C09146=1167.834,261.532,-67.033,-177.260,7.589,148.648
C09147=1167.838,261.283,-67.006,-177.262,7.587,148.648
C09148=1167.844,261.034,-66.978,-177.265,7.584,148.648
C09149=1167.847,260.786,-66.950,-177.268,7.581,148.649
C09150=1167.852,260.537,-66.922,-177.270,7.578,148.649
C09151=1167.856,260.290,-66.895,-177.273,7.575,148.649
C09152=1167.860,260.041,-66.867,-177.275,7.573,148.649
C09153=1167.865,259.792,-66.839,-177.278,7.570,148.649
C09154=1167.870,259.544,-66.811,-177.281,7.567,148.649
C09155=1167.874,259.296,-66.783,-177.284,7.564,148.649
C09156=1167.878,259.047,-66.756,-177.287,7.561,148.649
C09157=1167.883,258.799,-66.728,-177.289,7.559,148.649
C09158=1167.887,258.550,-66.701,-177.292,7.556,148.649
C09159=1167.891,258.302,-66.673,-177.295,7.553,148.649
C09160=1167.896,258.053,-66.645,-177.297,7.550,148.649
C09161=1167.900,257.805,-66.617,-177.299,7.548,148.650
C09162=1167.905,257.556,-66.590,-177.302,7.545,148.650
C09163=1167.909,257.309,-66.562,-177.305,7.542,148.650
C09164=1167.913,257.059,-66.535,-177.308,7.539,148.650
C09165=1167.917,256.811,-66.507,-177.310,7.537,148.650
C09166=1167.922,256.563,-66.480,-177.313,7.534,148.650
C09167=1167.926,256.314,-66.452,-177.316,7.531,148.650
C09168=1167.931,256.066,-66.425,-177.319,7.528,148.650
C09169=1167.935,255.818,-66.397,-177.321,7.526,148.650
C09170=1167.940,255.570,-66.370,-177.324,7.523,148.650
C09171=1167.944,255.320,-66.343,-177.326,7.520,148.650
C09172=1167.948,255.072,-66.315,-177.329,7.517,148.650
C09173=1167.953,254.824,-66.288,-177.331,7.515,148.651
C09174=1167.957,254.575,-66.260,-177.334,7.512,148.651
C09175=1167.961,254.327,-66.233,-177.337,7.510,148.651
C09176=1167.966,254.078,-66.205,-177.340,7.507,148.651
C09177=1167.970,253.830,-66.178,-177.342,7.505,148.651
C09178=1167.974,253.581,-66.150,-177.345,7.502,148.651
C09179=1167.979,253.333,-66.123,-177.348,7.499,148.651
C09180=1167.983,253.084,-66.096,-177.350,7.496,148.651
C09181=1167.988,252.836,-66.068,-177.353,7.494,148.651
C09182=1167.992,252.588,-66.041,-177.355,7.491,148.651
C09183=1167.996,252.339,-66.014,-177.359,7.488,148.652
C09184=1168.001,252.090,-65.987,-177.361,7.485,148.652
C09185=1168.005,251.842,-65.959,-177.364,7.483,148.652
C09186=1168.010,251.594,-65.932,-177.366,7.480,148.652
C09187=1168.014,251.346,-65.906,-177.369,7.477,148.652
C09188=1168.018,251.096,-65.878,-177.371,7.475,148.652
C09189=1168.023,250.848,-65.851,-177.375,7.472,148.652
C09190=1168.027,250.599,-65.824,-177.377,7.469,148.652
C09191=1168.032,250.352,-65.796,-177.380,7.466,148.652
C09192=1168.036,250.103,-65.769,-177.382,7.464,148.653
C09193=1168.041,249.855,-65.742,-177.385,7.461,148.653
C09194=1168.044,249.606,-65.715,-177.388,7.458,148.653
C09195=1168.049,249.357,-65.688,-177.390,7.457,148.653
C09196=1168.054,249.109,-65.661,-177.393,7.454,148.653
C09197=1168.058,248.860,-65.634,-177.396,7.451,148.653
C09198=1168.063,248.612,-65.607,-177.399,7.448,148.653
C09199=1168.067,248.364,-65.581,-177.401,7.446,148.653
C09200=1168.072,248.115,-65.553,-177.404,7.443,148.654
C09201=1168.076,247.866,-65.526,-177.407,7.440,148.654
C09202=1168.080,247.617,-65.499,-177.409,7.438,148.654
C09203=1168.084,247.369,-65.472,-177.412,7.435,148.654
C09204=1168.089,247.121,-65.445,-177.415,7.432,148.654
C09205=1168.094,246.872,-65.418,-177.417,7.430,148.654
C09206=1168.098,246.624,-65.391,-177.420,7.427,148.654
C09207=1168.102,246.376,-65.365,-177.423,7.424,148.654
C09208=1168.107,246.127,-65.338,-177.425,7.421,148.654
C09209=1168.111,245.879,-65.311,-177.428,7.419,148.655
C09210=1168.116,245.630,-65.284,-177.431,7.416,148.655
C09211=1168.120,245.382,-65.257,-177.434,7.413,148.655
C09212=1168.125,245.133,-65.231,-177.436,7.411,148.655
C09213=1168.129,244.884,-65.203,-177.439,7.408,148.655
C09214=1168.133,244.635,-65.177,-177.442,7.406,148.655
C09215=1168.138,244.387,-65.150,-177.444,7.404,148.655
C09216=1168.142,244.138,-65.123,-177.447,7.401,148.655
C09217=1168.146,243.890,-65.096,-177.449,7.398,148.656
C09218=1168.151,243.641,-65.070,-177.452,7.396,148.656
C09219=1168.155,243.393,-65.044,-177.455,7.393,148.656
C09220=1168.160,243.144,-65.016,-177.458,7.390,148.656
C09221=1168.164,242.896,-64.989,-177.460,7.388,148.656
C09222=1168.169,242.647,-64.964,-177.463,7.385,148.656
C09223=1168.173,242.399,-64.937,-177.466,7.382,148.656
C09224=1168.177,242.150,-64.910,-177.468,7.380,148.657
C09225=1168.182,241.901,-64.884,-177.471,7.377,148.657
C09226=1168.186,241.653,-64.857,-177.474,7.375,148.657
C09227=1168.191,241.405,-64.830,-177.476,7.372,148.657
C09228=1168.195,241.156,-64.803,-177.479,7.370,148.657
C09229=1168.200,240.907,-64.777,-177.482,7.367,148.657
C09230=1168.204,240.659,-64.750,-177.484,7.365,148.658
C09231=1168.208,240.410,-64.725,-177.487,7.362,148.658
C09232=1168.213,240.162,-64.698,-177.490,7.359,148.658
C09233=1168.217,239.913,-64.671,-177.493,7.357,148.658
C09234=1168.222,239.664,-64.645,-177.495,7.354,148.658
C09235=1168.227,239.417,-64.619,-177.497,7.352,148.658
C09236=1168.232,239.168,-64.592,-177.500,7.349,148.658
C09237=1168.235,238.919,-64.566,-177.503,7.346,148.659
C09238=1168.240,238.670,-64.540,-177.506,7.344,148.659
C09239=1168.244,238.422,-64.513,-177.508,7.341,148.659
C09240=1168.249,238.173,-64.487,-177.512,7.339,148.659
C09241=1168.253,237.925,-64.460,-177.514,7.337,148.659
C09242=1168.257,237.676,-64.434,-177.517,7.334,148.659
C09243=1168.262,237.428,-64.407,-177.520,7.331,148.659
C09244=1168.266,237.179,-64.382,-177.522,7.329,148.660
C09245=1168.271,236.930,-64.355,-177.525,7.326,148.660
C09246=1168.275,236.681,-64.329,-177.527,7.324,148.660
C09247=1168.280,236.411,-64.300,-177.530,7.321,148.660
C09248=1168.286,236.139,-64.272,-177.533,7.318,148.660
C09249=1168.290,235.867,-64.243,-177.536,7.316,148.660
C09250=1168.295,235.595,-64.214,-177.539,7.313,148.660
C09251=1168.299,235.347,-64.188,-177.542,7.310,148.661
C09252=1168.304,235.098,-64.162,-177.544,7.308,148.661
C09253=1168.309,234.849,-64.136,-177.547,7.305,148.661
C09254=1168.312,234.601,-64.109,-177.550,7.302,148.661
C09255=1168.317,234.352,-64.084,-177.553,7.300,148.661
C09256=1168.322,234.104,-64.058,-177.555,7.297,148.661
C09257=1168.326,233.855,-64.031,-177.558,7.295,148.662
C09258=1168.330,233.607,-64.005,-177.561,7.293,148.662
C09259=1168.335,233.358,-63.980,-177.563,7.290,148.662
C09260=1168.339,233.109,-63.953,-177.566,7.288,148.662
C09261=1168.344,232.861,-63.927,-177.569,7.285,148.662
C09262=1168.348,232.612,-63.902,-177.571,7.283,148.662
C09263=1168.353,232.363,-63.875,-177.574,7.280,148.663
C09264=1168.357,232.115,-63.849,-177.577,7.277,148.663
C09265=1168.361,231.866,-63.823,-177.580,7.275,148.663
C09266=1168.366,231.618,-63.798,-177.582,7.272,148.663
C09267=1168.370,231.369,-63.772,-177.585,7.270,148.663
C09268=1168.375,231.120,-63.745,-177.588,7.268,148.664
C09269=1168.380,230.871,-63.720,-177.591,7.265,148.664
C09270=1168.384,230.623,-63.694,-177.593,7.263,148.664
C09271=1168.389,230.375,-63.669,-177.596,7.260,148.664
C09272=1168.393,230.126,-63.642,-177.598,7.258,148.664
C09273=1168.398,229.877,-63.616,-177.602,7.255,148.664
C09274=1168.402,229.628,-63.590,-177.604,7.253,148.665
C09275=1168.407,229.380,-63.565,-177.606,7.250,148.665
C09276=1168.411,229.132,-63.539,-177.610,7.247,148.665
C09277=1168.415,228.883,-63.513,-177.612,7.245,148.665
C09278=1168.420,228.635,-63.488,-177.615,7.243,148.665
C09279=1168.424,228.386,-63.462,-177.617,7.241,148.665
C09280=1168.429,228.137,-63.436,-177.620,7.238,148.666
C09281=1168.433,227.888,-63.410,-177.623,7.236,148.666
C09282=1168.438,227.640,-63.385,-177.625,7.233,148.666
C09283=1168.442,227.391,-63.359,-177.628,7.231,148.666
C09284=1168.447,227.142,-63.333,-177.631,7.228,148.666
C09285=1168.451,226.894,-63.308,-177.634,7.225,148.666
C09286=1168.456,226.645,-63.282,-177.636,7.223,148.667
C09287=1168.460,226.397,-63.256,-177.639,7.220,148.667
C09288=1168.465,226.148,-63.231,-177.642,7.219,148.667
C09289=1168.469,225.899,-63.206,-177.645,7.216,148.667
C09290=1168.473,225.650,-63.180,-177.647,7.214,148.668
C09291=1168.478,225.402,-63.155,-177.650,7.211,148.668
C09292=1168.482,225.153,-63.129,-177.652,7.209,148.668
C09293=1168.487,224.904,-63.103,-177.655,7.206,148.668
C09294=1168.492,224.656,-63.078,-177.658,7.204,148.668
C09295=1168.496,224.408,-63.052,-177.661,7.202,148.669
C09296=1168.500,224.158,-63.027,-177.663,7.199,148.669
C09297=1168.505,223.910,-63.002,-177.666,7.197,148.669
C09298=1168.509,223.661,-62.976,-177.668,7.195,148.669
C09299=1168.514,223.413,-62.950,-177.672,7.192,148.669
C09300=1168.519,223.164,-62.925,-177.674,7.190,148.669
C09301=1168.523,222.915,-62.900,-177.677,7.187,148.670
C09302=1168.528,222.667,-62.874,-177.680,7.184,148.670
C09303=1168.532,222.418,-62.848,-177.682,7.182,148.670
C09304=1168.537,222.169,-62.824,-177.685,7.180,148.670
C09305=1168.541,221.920,-62.798,-177.687,7.178,148.670
C09306=1168.546,221.672,-62.772,-177.691,7.175,148.671
C09307=1168.550,221.423,-62.748,-177.693,7.173,148.671
C09308=1168.554,221.174,-62.722,-177.696,7.170,148.671
C09309=1168.559,220.926,-62.697,-177.698,7.168,148.671
C09310=1168.564,220.677,-62.672,-177.702,7.165,148.672
C09311=1168.568,220.429,-62.647,-177.704,7.163,148.672
C09312=1168.573,220.180,-62.621,-177.707,7.161,148.672
C09313=1168.577,219.931,-62.596,-177.709,7.159,148.672
C09314=1168.581,219.683,-62.571,-177.712,7.156,148.672
C09315=1168.586,219.433,-62.546,-177.715,7.154,148.673
C09316=1168.591,219.185,-62.521,-177.718,7.151,148.673
C09317=1168.595,218.936,-62.496,-177.720,7.149,148.673
C09318=1168.600,218.688,-62.470,-177.723,7.146,148.673
C09319=1168.604,218.439,-62.446,-177.725,7.144,148.673
C09320=1168.609,218.191,-62.420,-177.728,7.143,148.674
C09321=1168.613,217.941,-62.395,-177.731,7.140,148.674
C09322=1168.618,217.693,-62.370,-177.734,7.138,148.674
C09323=1168.622,217.444,-62.345,-177.736,7.135,148.674
C09324=1168.627,217.196,-62.320,-177.739,7.133,148.675
C09325=1168.631,216.946,-62.295,-177.742,7.130,148.675
C09326=1168.636,216.698,-62.270,-177.744,7.128,148.675
C09327=1168.640,216.449,-62.245,-177.747,7.125,148.675
C09328=1168.644,216.201,-62.220,-177.750,7.124,148.675
C09329=1168.649,215.952,-62.195,-177.753,7.121,148.675
C09330=1168.654,215.703,-62.170,-177.755,7.119,148.676
C09331=1168.658,215.454,-62.145,-177.758,7.116,148.676
C09332=1168.663,215.206,-62.120,-177.761,7.114,148.676
C09333=1168.668,214.958,-62.095,-177.764,7.111,148.676
C09334=1168.671,214.708,-62.071,-177.766,7.109,148.677
C09335=1168.677,214.460,-62.046,-177.768,7.107,148.677
C09336=1168.681,214.211,-62.020,-177.772,7.105,148.677
C09337=1168.685,213.963,-61.996,-177.774,7.103,148.677
C09338=1168.690,213.713,-61.971,-177.777,7.100,148.678
C09339=1168.695,213.464,-61.946,-177.780,7.098,148.678
C09340=1168.699,213.217,-61.922,-177.782,7.095,148.678
C09341=1168.703,212.967,-61.897,-177.785,7.094,148.678
C09342=1168.708,212.719,-61.872,-177.788,7.091,148.678
C09343=1168.712,212.469,-61.847,-177.791,7.089,148.679
C09344=1168.717,212.221,-61.822,-177.793,7.087,148.679
C09345=1168.722,211.973,-61.798,-177.796,7.084,148.679
C09346=1168.726,211.723,-61.773,-177.798,7.082,148.679
C09347=1168.730,211.475,-61.749,-177.801,7.079,148.680
C09348=1168.736,211.226,-61.724,-177.804,7.078,148.680
C09349=1168.739,210.977,-61.700,-177.807,7.075,148.680
C09350=1168.744,210.729,-61.674,-177.810,7.073,148.680
C09351=1168.749,210.458,-61.647,-177.812,7.070,148.680
C09352=1168.754,210.187,-61.621,-177.815,7.068,148.681
C09353=1168.759,209.917,-61.595,-177.818,7.065,148.681
C09354=1168.764,209.646,-61.568,-177.821,7.063,148.681
C09355=1168.768,209.398,-61.543,-177.824,7.061,148.682
C09356=1168.773,209.149,-61.519,-177.827,7.058,148.682
C09357=1168.777,208.900,-61.494,-177.829,7.056,148.682
C09358=1168.782,208.651,-61.470,-177.832,7.053,148.682
C09359=1168.787,208.403,-61.446,-177.835,7.051,148.682
C09360=1168.791,208.153,-61.421,-177.837,7.050,148.683
C09361=1168.796,207.905,-61.396,-177.840,7.047,148.683
C09362=1168.801,207.656,-61.372,-177.843,7.045,148.683
C09363=1168.805,207.408,-61.348,-177.846,7.042,148.684
C09364=1168.810,207.159,-61.323,-177.848,7.040,148.684
C09365=1168.814,206.910,-61.299,-177.851,7.038,148.684
C09366=1168.819,206.662,-61.275,-177.854,7.036,148.684
C09367=1168.824,206.413,-61.250,-177.856,7.034,148.684
C09368=1168.827,206.164,-61.225,-177.859,7.031,148.685
C09369=1168.833,205.915,-61.201,-177.862,7.029,148.685
C09370=1168.837,205.667,-61.177,-177.864,7.027,148.685
C09371=1168.841,205.418,-61.153,-177.868,7.024,148.686
C09372=1168.846,205.169,-61.128,-177.870,7.022,148.686
C09373=1168.850,204.920,-61.104,-177.872,7.021,148.686
C09374=1168.855,204.671,-61.080,-177.875,7.018,148.686
C09375=1168.860,204.423,-61.055,-177.878,7.016,148.686
C09376=1168.864,204.174,-61.031,-177.881,7.013,148.687
C09377=1168.868,203.925,-61.007,-177.883,7.011,148.687
C09378=1168.873,203.676,-60.982,-177.886,7.009,148.687
C09379=1168.878,203.427,-60.959,-177.889,7.007,148.688
C09380=1168.882,203.178,-60.934,-177.891,7.005,148.688
C09381=1168.887,202.930,-60.910,-177.894,7.003,148.688
C09382=1168.892,202.681,-60.886,-177.897,7.000,148.688
C09383=1168.896,202.433,-60.862,-177.900,6.998,148.688
C09384=1168.901,202.184,-60.838,-177.903,6.996,148.689
C09385=1168.905,201.934,-60.813,-177.905,6.993,148.689
C09386=1168.910,201.686,-60.789,-177.908,6.992,148.689
C09387=1168.914,201.437,-60.766,-177.911,6.989,148.690
C09388=1168.919,201.188,-60.742,-177.913,6.987,148.690
C09389=1168.924,200.940,-60.717,-177.916,6.985,148.690
C09390=1168.928,200.691,-60.694,-177.919,6.983,148.690
C09391=1168.932,200.442,-60.669,-177.921,6.980,148.691
C09392=1168.937,200.193,-60.645,-177.924,6.979,148.691
C09393=1168.941,199.944,-60.622,-177.927,6.976,148.691
C09394=1168.946,199.695,-60.597,-177.929,6.974,148.691
C09395=1168.951,199.446,-60.574,-177.932,6.972,148.692
C09396=1168.956,199.198,-60.550,-177.935,6.969,148.692
C09397=1168.960,198.950,-60.526,-177.937,6.967,148.692
C09398=1168.965,198.701,-60.502,-177.940,6.966,148.692
C09399=1168.968,198.451,-60.478,-177.943,6.963,148.693
C09400=1168.974,198.202,-60.454,-177.946,6.961,148.693
C09401=1168.978,197.954,-60.430,-177.948,6.959,148.693
C09402=1168.983,197.705,-60.407,-177.951,6.956,148.693
C09403=1168.987,197.456,-60.382,-177.954,6.954,148.694
C09404=1168.992,197.207,-60.359,-177.956,6.953,148.694
C09405=1168.996,196.959,-60.335,-177.959,6.950,148.694
C09406=1169.001,196.710,-60.312,-177.962,6.948,148.695
C09407=1169.006,196.461,-60.288,-177.965,6.946,148.695
C09408=1169.010,196.212,-60.264,-177.968,6.944,148.695
C09409=1169.015,195.964,-60.240,-177.970,6.942,148.695
C09410=1169.019,195.715,-60.217,-177.973,6.940,148.696
C09411=1169.024,195.465,-60.192,-177.976,6.937,148.696
C09412=1169.029,195.216,-60.168,-177.978,6.935,148.696
C09413=1169.033,194.967,-60.145,-177.981,6.933,148.697
C09414=1169.038,194.719,-60.121,-177.984,6.931,148.697
C09415=1169.042,194.470,-60.098,-177.986,6.929,148.697
C09416=1169.047,194.221,-60.074,-177.989,6.927,148.697
C09417=1169.051,193.972,-60.050,-177.992,6.924,148.698
C09418=1169.056,193.723,-60.027,-177.995,6.922,148.698
C09419=1169.061,193.474,-60.003,-177.997,6.920,148.698
C09420=1169.065,193.226,-59.979,-178.000,6.919,148.698
C09421=1169.070,192.977,-59.956,-178.003,6.916,148.699
C09422=1169.075,192.728,-59.933,-178.005,6.914,148.699
C09423=1169.079,192.479,-59.909,-178.008,6.912,148.699
C09424=1169.084,192.230,-59.885,-178.011,6.909,148.700
C09425=1169.088,191.982,-59.862,-178.013,6.907,148.700
C09426=1169.092,191.733,-59.839,-178.016,6.906,148.700
C09427=1169.097,191.484,-59.816,-178.019,6.903,148.700
C09428=1169.102,191.235,-59.792,-178.022,6.901,148.701
C09429=1169.106,190.986,-59.768,-178.024,6.899,148.701
C09430=1169.111,190.737,-59.745,-178.027,6.897,148.701
C09431=1169.116,190.489,-59.722,-178.030,6.895,148.702
C09432=1169.121,190.240,-59.699,-178.033,6.893,148.702
C09433=1169.126,189.991,-59.675,-178.035,6.891,148.702
C09434=1169.130,189.742,-59.651,-178.038,6.889,148.702
C09435=1169.135,189.493,-59.628,-178.041,6.886,148.703
C09436=1169.139,189.245,-59.605,-178.043,6.885,148.703
C09437=1169.143,188.996,-59.582,-178.046,6.883,148.703
C09438=1169.148,188.747,-59.558,-178.049,6.880,148.704
C09439=1169.153,188.498,-59.535,-178.052,6.878,148.704
C09440=1169.157,188.249,-59.512,-178.054,6.876,148.704
C09441=1169.162,187.999,-59.488,-178.056,6.874,148.704
C09442=1169.166,187.751,-59.465,-178.060,6.872,148.705
C09443=1169.171,187.502,-59.442,-178.062,6.870,148.705
C09444=1169.176,187.253,-59.419,-178.065,6.868,148.705
C09445=1169.181,187.004,-59.396,-178.067,6.866,148.706
C09446=1169.186,186.755,-59.372,-178.071,6.864,148.706
C09447=1169.189,186.507,-59.350,-178.073,6.862,148.706
C09448=1169.194,186.258,-59.326,-178.076,6.860,148.707
C09449=1169.199,186.009,-59.303,-178.078,6.858,148.707
C09450=1169.204,185.760,-59.280,-178.081,6.855,148.707
C09451=1169.208,185.512,-59.257,-178.084,6.854,148.707
C09452=1169.213,185.262,-59.234,-178.087,6.852,148.708
C09453=1169.218,185.013,-59.210,-178.089,6.850,148.708
C09454=1169.222,184.765,-59.188,-178.092,6.847,148.708
C09455=1169.227,184.495,-59.163,-178.095,6.845,148.709
C09456=1169.232,184.225,-59.138,-178.098,6.843,148.709
C09457=1169.237,183.956,-59.113,-178.101,6.841,148.709
C09458=1169.242,183.686,-59.088,-178.104,6.838,148.710
C09459=1169.247,183.437,-59.065,-178.107,6.837,148.710
C09460=1169.251,183.188,-59.042,-178.109,6.834,148.710
C09461=1169.255,182.939,-59.019,-178.112,6.833,148.711
C09462=1169.261,182.691,-58.996,-178.114,6.831,148.711
C09463=1169.265,182.442,-58.974,-178.118,6.828,148.711
C09464=1169.270,182.192,-58.950,-178.120,6.827,148.712
C09465=1169.274,181.943,-58.927,-178.122,6.824,148.712
C09466=1169.278,181.695,-58.904,-178.125,6.823,148.712
C09467=1169.284,181.446,-58.882,-178.128,6.820,148.712
C09468=1169.288,181.197,-58.859,-178.131,6.818,148.713
C09469=1169.293,180.948,-58.836,-178.134,6.817,148.713
C09470=1169.297,180.699,-58.812,-178.136,6.814,148.713
C09471=1169.302,180.450,-58.791,-178.139,6.813,148.714
C09472=1169.307,180.201,-58.767,-178.142,6.810,148.714
C09473=1169.311,179.953,-58.745,-178.145,6.808,148.714
C09474=1169.316,179.703,-58.722,-178.147,6.807,148.715
C09475=1169.320,179.455,-58.700,-178.150,6.805,148.715
C09476=1169.325,179.206,-58.676,-178.152,6.803,148.715
C09477=1169.329,178.957,-58.654,-178.155,6.800,148.716
C09478=1169.334,178.708,-58.631,-178.158,6.798,148.716
C09479=1169.339,178.460,-58.608,-178.161,6.797,148.716
C09480=1169.344,178.210,-58.586,-178.163,6.795,148.717
C09481=1169.348,177.961,-58.563,-178.166,6.793,148.717
C09482=1169.353,177.712,-58.541,-178.169,6.790,148.717
C09483=1169.357,177.463,-58.518,-178.172,6.788,148.718
C09484=1169.362,177.214,-58.495,-178.174,6.787,148.718
C09485=1169.367,176.966,-58.473,-178.177,6.785,148.718
C09486=1169.372,176.716,-58.450,-178.180,6.783,148.719
C09487=1169.376,176.467,-58.427,-178.182,6.781,148.719
C09488=1169.381,176.218,-58.405,-178.185,6.778,148.719
C09489=1169.385,175.970,-58.382,-178.188,6.777,148.719
C09490=1169.390,175.720,-58.360,-178.190,6.775,148.720
C09491=1169.395,175.472,-58.337,-178.193,6.773,148.720
C09492=1169.399,175.223,-58.315,-178.196,6.771,148.721
C09493=1169.404,174.974,-58.292,-178.199,6.769,148.721
C09494=1169.409,174.725,-58.270,-178.201,6.767,148.721
C09495=1169.413,174.476,-58.247,-178.204,6.765,148.721
C09496=1169.418,174.227,-58.225,-178.207,6.763,148.722
C09497=1169.423,173.978,-58.203,-178.209,6.761,148.722
C09498=1169.427,173.729,-58.180,-178.212,6.760,148.722
C09499=1169.432,173.480,-58.158,-178.215,6.758,148.723
C09500=1169.437,173.231,-58.135,-178.218,6.755,148.723
C09501=1169.441,172.982,-58.113,-178.220,6.753,148.723
C09502=1169.446,172.733,-58.091,-178.223,6.751,148.724
C09503=1169.451,172.484,-58.068,-178.226,6.750,148.724
C09504=1169.455,172.235,-58.046,-178.228,6.748,148.724
C09505=1169.460,171.986,-58.024,-178.231,6.746,148.725
C09506=1169.464,171.737,-58.001,-178.234,6.744,148.725
C09507=1169.469,171.489,-57.979,-178.237,6.742,148.726
C09508=1169.474,171.239,-57.957,-178.240,6.740,148.726
C09509=1169.478,170.991,-57.935,-178.242,6.738,148.726
C09510=1169.483,170.742,-57.912,-178.244,6.736,148.726
C09511=1169.487,170.492,-57.890,-178.247,6.734,148.727
C09512=1169.492,170.244,-57.868,-178.250,6.733,148.727
C09513=1169.497,169.994,-57.845,-178.253,6.731,148.727
C09514=1169.502,169.746,-57.823,-178.256,6.728,148.728
C09515=1169.506,169.497,-57.801,-178.258,6.727,148.728
C09516=1169.511,169.248,-57.779,-178.261,6.725,148.729
C09517=1169.515,168.999,-57.757,-178.264,6.723,148.729
C09518=1169.521,168.750,-57.735,-178.266,6.721,148.729
C09519=1169.525,168.500,-57.713,-178.269,6.719,148.729
C09520=1169.530,168.252,-57.691,-178.271,6.717,148.730
C09521=1169.534,168.003,-57.669,-178.274,6.716,148.730
C09522=1169.540,167.754,-57.646,-178.277,6.713,148.731
C09523=1169.544,167.505,-57.624,-178.280,6.711,148.731
C09524=1169.549,167.256,-57.603,-178.283,6.710,148.731
C09525=1169.553,167.007,-57.580,-178.285,6.708,148.732
C09526=1169.558,166.758,-57.559,-178.288,6.706,148.732
C09527=1169.562,166.509,-57.537,-178.291,6.704,148.732
C09528=1169.568,166.260,-57.514,-178.294,6.703,148.733
C09529=1169.572,166.010,-57.492,-178.296,6.700,148.733
C09530=1169.577,165.762,-57.471,-178.298,6.699,148.733
C09531=1169.581,165.512,-57.449,-178.302,6.696,148.734
C09532=1169.586,165.264,-57.427,-178.304,6.694,148.734
C09533=1169.590,165.015,-57.405,-178.307,6.693,148.734
C09534=1169.595,164.766,-57.383,-178.310,6.691,148.735
C09535=1169.599,164.517,-57.361,-178.312,6.689,148.735
C09536=1169.604,164.268,-57.340,-178.315,6.687,148.735
C09537=1169.609,164.019,-57.318,-178.318,6.686,148.736
C09538=1169.613,163.770,-57.296,-178.321,6.684,148.736
C09539=1169.618,163.521,-57.274,-178.323,6.682,148.737
C09540=1169.623,163.272,-57.251,-178.326,6.680,148.737
C09541=1169.628,163.023,-57.230,-178.329,6.679,148.737
C09542=1169.632,162.774,-57.208,-178.332,6.676,148.738
C09543=1169.637,162.525,-57.186,-178.335,6.674,148.738
C09544=1169.642,162.276,-57.165,-178.337,6.672,148.738
C09545=1169.647,162.026,-57.143,-178.339,6.670,148.739
C09546=1169.652,161.778,-57.121,-178.342,6.669,148.739
C09547=1169.657,161.529,-57.100,-178.345,6.667,148.739
C09548=1169.661,161.280,-57.078,-178.348,6.665,148.740
C09549=1169.666,161.031,-57.056,-178.350,6.663,148.740
C09550=1169.670,160.781,-57.035,-178.353,6.662,148.740
C09551=1169.675,160.533,-57.013,-178.356,6.660,148.741
C09552=1169.679,160.284,-56.992,-178.358,6.658,148.741
C09553=1169.683,160.035,-56.970,-178.361,6.656,148.742
C09554=1169.688,159.786,-56.948,-178.364,6.655,148.742
C09555=1169.694,159.537,-56.927,-178.366,6.653,148.742
C09556=1169.698,159.288,-56.905,-178.369,6.651,148.743
C09557=1169.703,159.039,-56.883,-178.372,6.648,148.743
C09558=1169.708,158.790,-56.862,-178.375,6.647,148.743
C09559=1169.713,158.521,-56.838,-178.378,6.645,148.744
C09560=1169.718,158.252,-56.816,-178.380,6.643,148.744
C09561=1169.723,157.983,-56.792,-178.383,6.641,148.745
C09562=1169.728,157.714,-56.769,-178.386,6.639,148.745
C09563=1169.733,157.465,-56.748,-178.389,6.637,148.745
C09564=1169.737,157.216,-56.726,-178.392,6.635,148.746
C09565=1169.742,156.966,-56.705,-178.394,6.634,148.746
C09566=1169.747,156.718,-56.683,-178.397,6.632,148.746
C09567=1169.751,156.469,-56.662,-178.400,6.630,148.747
C09568=1169.756,156.219,-56.641,-178.402,6.628,148.747
C09569=1169.761,155.971,-56.619,-178.405,6.627,148.748
C09570=1169.766,155.721,-56.598,-178.408,6.625,148.748
C09571=1169.770,155.472,-56.576,-178.411,6.623,148.748
C09572=1169.774,155.224,-56.555,-178.413,6.621,148.749
C09573=1169.780,154.975,-56.534,-178.416,6.620,148.749
C09574=1169.784,154.726,-56.512,-178.419,6.618,148.749
C09575=1169.789,154.476,-56.491,-178.421,6.616,148.750
C09576=1169.794,154.227,-56.469,-178.424,6.614,148.750
C09577=1169.798,153.978,-56.449,-178.427,6.613,148.751
C09578=1169.803,153.730,-56.427,-178.429,6.611,148.751
C09579=1169.808,153.480,-56.406,-178.432,6.609,148.751
C09580=1169.813,153.231,-56.384,-178.435,6.607,148.752
C09581=1169.817,152.982,-56.364,-178.438,6.606,148.752
C09582=1169.822,152.733,-56.343,-178.440,6.604,148.752
C09583=1169.826,152.484,-56.321,-178.443,6.602,148.753
C09584=1169.832,152.234,-56.300,-178.446,6.600,148.753
C09585=1169.836,151.986,-56.279,-178.448,6.599,148.754
C09586=1169.841,151.737,-56.258,-178.451,6.597,148.754
C09587=1169.846,151.487,-56.237,-178.454,6.595,148.754
C09588=1169.850,151.239,-56.216,-178.456,6.593,148.755
C09589=1169.855,150.989,-56.194,-178.460,6.592,148.755
C09590=1169.860,150.740,-56.173,-178.462,6.590,148.756
C09591=1169.864,150.492,-56.152,-178.465,6.589,148.756
C09592=1169.869,150.242,-56.131,-178.468,6.587,148.756
C09593=1169.874,149.993,-56.110,-178.470,6.585,148.757
C09594=1169.879,149.745,-56.089,-178.473,6.583,148.757
C09595=1169.883,149.495,-56.068,-178.476,6.582,148.758
C09596=1169.888,149.245,-56.047,-178.478,6.580,148.758
C09597=1169.892,148.997,-56.026,-178.481,6.578,148.758
C09598=1169.898,148.748,-56.005,-178.484,6.576,148.759
C09599=1169.902,148.499,-55.985,-178.486,6.575,148.759
C09600=1169.907,148.250,-55.964,-178.489,6.573,148.760
C09601=1169.912,148.001,-55.942,-178.492,6.571,148.760
C09602=1169.916,147.751,-55.921,-178.495,6.569,148.760
C09603=1169.921,147.502,-55.900,-178.497,6.568,148.761
C09604=1169.926,147.253,-55.880,-178.500,6.566,148.761
C09605=1169.931,147.004,-55.859,-178.503,6.564,148.761
C09606=1169.936,146.755,-55.837,-178.505,6.562,148.762
C09607=1169.940,146.506,-55.817,-178.508,6.561,148.762
C09608=1169.945,146.257,-55.796,-178.511,6.559,148.763
C09609=1169.950,146.008,-55.776,-178.513,6.557,148.763
C09610=1169.955,145.759,-55.755,-178.516,6.555,148.763
C09611=1169.959,145.510,-55.734,-178.519,6.554,148.764
C09612=1169.964,145.261,-55.713,-178.522,6.552,148.764
C09613=1169.968,145.011,-55.692,-178.525,6.550,148.765
C09614=1169.973,144.762,-55.671,-178.527,6.549,148.765
C09615=1169.978,144.513,-55.650,-178.530,6.547,148.765
C09616=1169.983,144.264,-55.629,-178.532,6.546,148.766
C09617=1169.987,144.015,-55.609,-178.535,6.544,148.766
C09618=1169.992,143.766,-55.588,-178.538,6.543,148.767
C09619=1169.997,143.517,-55.568,-178.540,6.541,148.767
C09620=1170.001,143.268,-55.547,-178.543,6.539,148.767
C09621=1170.006,143.019,-55.526,-178.546,6.537,148.768
C09622=1170.011,142.770,-55.506,-178.548,6.536,148.768
C09623=1170.016,142.521,-55.485,-178.551,6.534,148.769
C09624=1170.020,142.272,-55.465,-178.554,6.532,148.769
C09625=1170.025,142.023,-55.444,-178.557,6.531,148.770
C09626=1170.030,141.773,-55.423,-178.560,6.529,148.770
C09627=1170.035,141.524,-55.403,-178.562,6.527,148.770
C09628=1170.040,141.275,-55.382,-178.565,6.526,148.771
C09629=1170.044,141.026,-55.362,-178.568,6.524,148.771
C09630=1170.049,140.777,-55.341,-178.571,6.522,148.771
C09631=1170.054,140.527,-55.321,-178.573,6.520,148.772
C09632=1170.058,140.278,-55.301,-178.575,6.519,148.772
C09633=1170.063,140.030,-55.280,-178.578,6.518,148.773
C09634=1170.068,139.780,-55.259,-178.581,6.516,148.773
C09635=1170.073,139.531,-55.239,-178.584,6.514,148.774
C09636=1170.077,139.282,-55.219,-178.587,6.513,148.774
C09637=1170.082,139.033,-55.198,-178.589,6.511,148.774
C09638=1170.087,138.784,-55.178,-178.592,6.509,148.775
C09639=1170.091,138.535,-55.158,-178.595,6.508,148.775
C09640=1170.097,138.285,-55.137,-178.597,6.506,148.776
C09641=1170.101,138.036,-55.116,-178.600,6.504,148.776
C09642=1170.105,137.787,-55.096,-178.603,6.502,148.776
C09643=1170.111,137.538,-55.076,-178.605,6.501,148.777
C09644=1170.116,137.289,-55.056,-178.608,6.500,148.777
C09645=1170.120,137.040,-55.035,-178.611,6.498,148.778
C09646=1170.125,136.791,-55.015,-178.614,6.497,148.778
C09647=1170.130,136.542,-54.995,-178.616,6.495,148.779
C09648=1170.135,136.293,-54.974,-178.619,6.493,148.779
C09649=1170.139,136.044,-54.954,-178.622,6.491,148.779
C09650=1170.144,135.794,-54.934,-178.624,6.490,148.780
C09651=1170.149,135.545,-54.913,-178.627,6.488,148.780
C09652=1170.153,135.296,-54.893,-178.630,6.487,148.781
C09653=1170.158,135.047,-54.872,-178.632,6.486,148.781
C09654=1170.163,134.798,-54.853,-178.635,6.484,148.782
C09655=1170.168,134.549,-54.833,-178.638,6.482,148.782
C09656=1170.173,134.299,-54.813,-178.640,6.480,148.782
C09657=1170.178,134.050,-54.792,-178.643,6.479,148.783
C09658=1170.182,133.801,-54.772,-178.646,6.477,148.783
C09659=1170.187,133.552,-54.752,-178.649,6.475,148.783
C09660=1170.191,133.303,-54.732,-178.651,6.475,148.784
C09661=1170.197,133.054,-54.713,-178.654,6.473,148.784
C09662=1170.201,132.805,-54.692,-178.657,6.471,148.785
C09663=1170.207,132.536,-54.670,-178.659,6.469,148.785
C09664=1170.211,132.268,-54.649,-178.662,6.468,148.786
C09665=1170.217,131.999,-54.627,-178.665,6.466,148.786
C09666=1170.222,131.730,-54.606,-178.668,6.464,148.787
C09667=1170.226,131.481,-54.586,-178.671,6.463,148.787
C09668=1170.232,131.232,-54.565,-178.673,6.461,148.787
C09669=1170.236,130.983,-54.545,-178.676,6.460,148.788
C09670=1170.242,130.734,-54.526,-178.679,6.458,148.788
C09671=1170.246,130.485,-54.505,-178.682,6.456,148.789
C09672=1170.251,130.235,-54.486,-178.685,6.454,148.789
C09673=1170.255,129.986,-54.465,-178.687,6.453,148.790
C09674=1170.260,129.737,-54.446,-178.689,6.452,148.790
C09675=1170.265,129.488,-54.426,-178.693,6.450,148.791
C09676=1170.270,129.239,-54.406,-178.695,6.449,148.791
C09677=1170.274,128.989,-54.386,-178.698,6.447,148.791
C09678=1170.279,128.740,-54.366,-178.701,6.445,148.792
C09679=1170.284,128.492,-54.347,-178.703,6.443,148.792
C09680=1170.289,128.243,-54.326,-178.706,6.443,148.793
C09681=1170.293,127.993,-54.307,-178.709,6.441,148.793
C09682=1170.298,127.743,-54.287,-178.711,6.439,148.794
C09683=1170.303,127.495,-54.267,-178.714,6.438,148.794
C09684=1170.308,127.246,-54.247,-178.717,6.436,148.794
C09685=1170.313,126.996,-54.228,-178.720,6.434,148.795
C09686=1170.317,126.747,-54.207,-178.722,6.434,148.795
C09687=1170.322,126.498,-54.188,-178.725,6.432,148.796
C09688=1170.327,126.249,-54.168,-178.728,6.430,148.796
C09689=1170.332,125.999,-54.149,-178.730,6.428,148.797
C09690=1170.337,125.751,-54.129,-178.733,6.427,148.797
C09691=1170.342,125.501,-54.109,-178.735,6.426,148.797
C09692=1170.346,125.252,-54.089,-178.738,6.424,148.798
C09693=1170.350,125.002,-54.070,-178.741,6.423,148.798
C09694=1170.355,124.754,-54.050,-178.744,6.421,148.799
C09695=1170.360,124.505,-54.031,-178.746,6.419,148.799
C09696=1170.365,124.255,-54.011,-178.749,6.418,148.800
C09697=1170.370,124.006,-53.992,-178.752,6.417,148.800
C09698=1170.375,123.757,-53.972,-178.754,6.415,148.801
C09699=1170.380,123.508,-53.952,-178.757,6.414,148.801
C09700=1170.385,123.259,-53.932,-178.760,6.412,148.801
C09701=1170.389,123.010,-53.913,-178.763,6.410,148.802
C09702=1170.394,122.760,-53.894,-178.765,6.410,148.803
C09703=1170.399,122.511,-53.874,-178.768,6.408,148.803
C09704=1170.404,122.262,-53.855,-178.771,6.406,148.803
C09705=1170.408,122.012,-53.835,-178.773,6.404,148.804
C09706=1170.413,121.764,-53.815,-178.776,6.403,148.804
C09707=1170.417,121.514,-53.796,-178.779,6.402,148.805
C09708=1170.423,121.266,-53.777,-178.781,6.400,148.805
C09709=1170.428,121.016,-53.757,-178.784,6.399,148.806
C09710=1170.432,120.766,-53.737,-178.787,6.397,148.806
C09711=1170.438,120.518,-53.718,-178.789,6.396,148.807
C09712=1170.442,120.268,-53.699,-178.792,6.395,148.807
C09713=1170.447,120.020,-53.680,-178.795,6.393,148.807
C09714=1170.452,119.770,-53.660,-178.797,6.391,148.808
C09715=1170.456,119.520,-53.640,-178.800,6.389,148.808
C09716=1170.461,119.272,-53.622,-178.803,6.389,148.809
C09717=1170.466,119.022,-53.602,-178.806,6.387,148.809
C09718=1170.471,118.773,-53.583,-178.808,6.385,148.810
C09719=1170.476,118.524,-53.563,-178.811,6.384,148.810
C09720=1170.480,118.275,-53.544,-178.814,6.383,148.811
C09721=1170.485,118.026,-53.525,-178.816,6.381,148.811
C09722=1170.490,117.776,-53.505,-178.819,6.380,148.811
C09723=1170.495,117.528,-53.486,-178.822,6.378,148.812
C09724=1170.500,117.277,-53.467,-178.824,6.377,148.812
C09725=1170.505,117.028,-53.448,-178.827,6.376,148.813
C09726=1170.509,116.779,-53.429,-178.830,6.374,148.813
C09727=1170.514,116.530,-53.410,-178.832,6.372,148.814
C09728=1170.519,116.281,-53.390,-178.835,6.372,148.814
C09729=1170.524,116.032,-53.371,-178.838,6.370,148.815
C09730=1170.528,115.783,-53.352,-178.840,6.368,148.815
C09731=1170.534,115.534,-53.332,-178.843,6.366,148.816
C09732=1170.538,115.284,-53.314,-178.846,6.366,148.816
C09733=1170.543,115.035,-53.295,-178.848,6.364,148.817
C09734=1170.548,114.785,-53.275,-178.851,6.362,148.817
C09735=1170.553,114.537,-53.256,-178.854,6.361,148.817
C09736=1170.558,114.287,-53.237,-178.857,6.360,148.818
C09737=1170.562,114.038,-53.219,-178.859,6.358,148.818
C09738=1170.567,113.789,-53.199,-178.862,6.357,148.819
C09739=1170.573,113.540,-53.180,-178.865,6.355,148.819
C09740=1170.577,113.291,-53.161,-178.867,6.354,148.820
C09741=1170.582,113.041,-53.142,-178.870,6.353,148.820
C09742=1170.586,112.792,-53.123,-178.873,6.351,148.821
C09743=1170.592,112.543,-53.104,-178.875,6.349,148.821
C09744=1170.596,112.293,-53.086,-178.878,6.349,148.822
C09745=1170.601,112.044,-53.066,-178.881,6.347,148.822
C09746=1170.606,111.795,-53.047,-178.883,6.345,148.823
C09747=1170.611,111.545,-53.029,-178.886,6.344,148.823
C09748=1170.616,111.297,-53.009,-178.889,6.343,148.824
C09749=1170.620,111.047,-52.990,-178.891,6.341,148.824
C09750=1170.626,110.798,-52.972,-178.894,6.340,148.824
C09751=1170.630,110.549,-52.953,-178.897,6.339,148.825
C09752=1170.635,110.300,-52.933,-178.900,6.337,148.825
C09753=1170.640,110.050,-52.915,-178.902,6.336,148.826
C09754=1170.645,109.801,-52.896,-178.904,6.335,148.826
C09755=1170.650,109.552,-52.878,-178.908,6.333,148.827
C09756=1170.655,109.302,-52.858,-178.910,6.332,148.827
C09757=1170.659,109.054,-52.839,-178.913,6.330,148.828
C09758=1170.663,108.804,-52.821,-178.916,6.329,148.828
C09759=1170.669,108.555,-52.802,-178.918,6.328,148.829
C09760=1170.674,108.306,-52.784,-178.921,6.326,148.829
C09761=1170.678,108.056,-52.764,-178.923,6.325,148.830
C09762=1170.683,107.807,-52.746,-178.926,6.324,148.830
C09763=1170.688,107.557,-52.726,-178.929,6.322,148.831
C09764=1170.693,107.308,-52.708,-178.931,6.321,148.831
C09765=1170.698,107.060,-52.690,-178.934,6.320,148.832
C09766=1170.703,106.809,-52.671,-178.937,6.318,148.832
C09767=1170.707,106.542,-52.651,-178.940,6.316,148.832
C09768=1170.713,106.273,-52.631,-178.943,6.315,148.833
C09769=1170.718,106.005,-52.611,-178.945,6.314,148.834
C09770=1170.723,105.736,-52.590,-178.948,6.313,148.834
C09771=1170.728,105.487,-52.572,-178.951,6.311,148.835
C09772=1170.734,105.238,-52.554,-178.954,6.309,148.835
C09773=1170.738,104.988,-52.535,-178.956,6.309,148.836
C09774=1170.743,104.739,-52.517,-178.959,6.307,148.836
C09775=1170.748,104.490,-52.497,-178.962,6.305,148.836
C09776=1170.752,104.241,-52.479,-178.964,6.305,148.837
C09777=1170.757,103.991,-52.461,-178.967,6.303,148.837
C09778=1170.763,103.742,-52.442,-178.970,6.301,148.838
C09779=1170.767,103.493,-52.423,-178.973,6.301,148.839
C09780=1170.772,103.243,-52.405,-178.975,6.299,148.839
C09781=1170.776,102.995,-52.387,-178.978,6.297,148.839
C09782=1170.782,102.745,-52.368,-178.981,6.297,148.840
C09783=1170.786,102.496,-52.350,-178.983,6.295,148.840
C09784=1170.791,102.247,-52.331,-178.986,6.293,148.841
C09785=1170.796,101.998,-52.313,-178.988,6.292,148.841
C09786=1170.802,101.748,-52.295,-178.991,6.291,148.842
C09787=1170.806,101.498,-52.276,-178.994,6.289,148.842
C09788=1170.811,101.250,-52.257,-178.996,6.288,148.843
C09789=1170.815,101.001,-52.240,-178.999,6.287,148.843
C09790=1170.820,100.750,-52.221,-179.002,6.285,148.844
C09791=1170.825,100.501,-52.203,-179.004,6.284,148.844
C09792=1170.830,100.252,-52.185,-179.007,6.283,148.845
C09793=1170.835,100.004,-52.166,-179.010,6.281,148.845
C09794=1170.840,99.754,-52.148,-179.012,6.280,148.846
C09795=1170.845,99.504,-52.129,-179.016,6.279,148.846
C09796=1170.850,99.255,-52.111,-179.018,6.278,148.847
C09797=1170.855,99.006,-52.093,-179.020,6.276,148.847
C09798=1170.859,98.757,-52.074,-179.024,6.275,148.848
C09799=1170.864,98.507,-52.056,-179.026,6.274,148.848
C09800=1170.869,98.258,-52.038,-179.028,6.273,148.849
C09801=1170.874,98.009,-52.019,-179.032,6.271,148.849
C09802=1170.879,97.760,-52.001,-179.034,6.270,148.850
C09803=1170.884,97.510,-51.983,-179.036,6.269,148.850
C09804=1170.888,97.261,-51.965,-179.039,6.268,148.851
C09805=1170.893,97.011,-51.947,-179.042,6.266,148.851
C09806=1170.898,96.762,-51.929,-179.045,6.265,148.852
C09807=1170.903,96.513,-51.911,-179.047,6.264,148.852
C09808=1170.908,96.264,-51.893,-179.050,6.262,148.853
C09809=1170.914,96.014,-51.875,-179.053,6.261,148.853
C09810=1170.918,95.765,-51.856,-179.055,6.260,148.854
C09811=1170.923,95.516,-51.838,-179.058,6.258,148.854
C09812=1170.927,95.267,-51.820,-179.061,6.258,148.855
C09813=1170.932,95.018,-51.802,-179.063,6.256,148.855
C09814=1170.937,94.768,-51.784,-179.066,6.254,148.856
C09815=1170.942,94.519,-51.766,-179.069,6.254,148.856
C09816=1170.947,94.269,-51.748,-179.071,6.252,148.857
C09817=1170.952,94.020,-51.730,-179.074,6.251,148.857
C09818=1170.957,93.770,-51.712,-179.077,6.250,148.858
C09819=1170.962,93.521,-51.694,-179.079,6.248,148.858
C09820=1170.966,93.272,-51.676,-179.082,6.248,148.859
C09821=1170.971,93.023,-51.658,-179.085,6.246,148.859
C09822=1170.976,92.774,-51.640,-179.087,6.245,148.860
C09823=1170.981,92.525,-51.622,-179.090,6.244,148.860
C09824=1170.986,92.275,-51.604,-179.093,6.242,148.861
C09825=1170.991,92.026,-51.586,-179.095,6.241,148.861
C09826=1170.996,91.777,-51.568,-179.098,6.240,148.862
C09827=1171.001,91.526,-51.551,-179.100,6.239,148.862
C09828=1171.005,91.277,-51.533,-179.104,6.238,148.863
C09829=1171.010,91.028,-51.515,-179.106,6.237,148.863
C09830=1171.015,90.779,-51.497,-179.108,6.235,148.864
C09831=1171.020,90.530,-51.479,-179.112,6.234,148.864
C09832=1171.025,90.281,-51.461,-179.114,6.233,148.865
C09833=1171.030,90.031,-51.443,-179.116,6.231,148.865
C09834=1171.035,89.782,-51.425,-179.119,6.230,148.866
C09835=1171.039,89.533,-51.408,-179.122,6.229,148.866
C09836=1171.044,89.284,-51.390,-179.125,6.227,148.867
C09837=1171.050,89.034,-51.373,-179.127,6.227,148.867
C09838=1171.054,88.785,-51.355,-179.130,6.225,148.868
C09839=1171.059,88.535,-51.337,-179.132,6.224,148.868
C09840=1171.064,88.286,-51.319,-179.135,6.223,148.869
C09841=1171.069,88.036,-51.302,-179.138,6.222,148.869
C09842=1171.074,87.787,-51.284,-179.141,6.220,148.870
C09843=1171.079,87.538,-51.266,-179.143,6.219,148.870
C09844=1171.084,87.289,-51.249,-179.146,6.218,148.871
C09845=1171.089,87.039,-51.231,-179.149,6.216,148.871
C09846=1171.094,86.790,-51.213,-179.151,6.216,148.872
C09847=1171.099,86.540,-51.196,-179.154,6.214,148.872
C09848=1171.104,86.291,-51.178,-179.156,6.213,148.873
C09849=1171.109,86.042,-51.160,-179.159,6.212,148.873
C09850=1171.113,85.793,-51.143,-179.161,6.211,148.874
C09851=1171.118,85.543,-51.125,-179.164,6.209,148.874
C09852=1171.123,85.294,-51.107,-179.167,6.209,148.875
C09853=1171.128,85.045,-51.090,-179.170,6.207,148.875
C09854=1171.132,84.796,-51.073,-179.172,6.207,148.876
C09855=1171.138,84.546,-51.055,-179.175,6.205,148.876
C09856=1171.142,84.297,-51.037,-179.178,6.204,148.877
C09857=1171.148,84.047,-51.020,-179.180,6.203,148.877
C09858=1171.153,83.798,-51.002,-179.183,6.201,148.878
C09859=1171.157,83.549,-50.985,-179.186,6.200,148.879
C09860=1171.162,83.299,-50.967,-179.188,6.199,148.879
C09861=1171.167,83.050,-50.949,-179.191,6.198,148.880
C09862=1171.171,82.800,-50.933,-179.194,6.196,148.880
C09863=1171.176,82.551,-50.915,-179.196,6.196,148.880
C09864=1171.182,82.302,-50.898,-179.199,6.194,148.881
C09865=1171.187,82.053,-50.880,-179.201,6.193,148.882
C09866=1171.191,81.803,-50.863,-179.204,6.192,148.882
C09867=1171.196,81.554,-50.845,-179.207,6.191,148.883
C09868=1171.202,81.304,-50.828,-179.210,6.190,148.883
C09869=1171.206,81.055,-50.811,-179.212,6.189,148.884
C09870=1171.211,80.806,-50.793,-179.215,6.187,148.884
C09871=1171.216,80.537,-50.775,-179.218,6.186,148.885
C09872=1171.222,80.269,-50.756,-179.220,6.185,148.885
C09873=1171.227,80.001,-50.738,-179.223,6.184,148.886
C09874=1171.232,79.732,-50.719,-179.226,6.182,148.887
C09875=1171.237,79.482,-50.702,-179.229,6.181,148.887
C09876=1171.242,79.234,-50.685,-179.232,6.180,148.888
C09877=1171.247,78.984,-50.667,-179.234,6.179,148.888
C09878=1171.253,78.734,-50.650,-179.237,6.178,148.889
C09879=1171.257,78.486,-50.633,-179.239,6.177,148.889
C09880=1171.262,78.236,-50.615,-179.242,6.175,148.890
C09881=1171.266,77.986,-50.599,-179.245,6.175,148.890
C09882=1171.272,77.738,-50.581,-179.247,6.173,148.891
C09883=1171.277,77.488,-50.564,-179.250,6.173,148.891
C09884=1171.282,77.239,-50.547,-179.253,6.171,148.892
C09885=1171.287,76.989,-50.529,-179.255,6.170,148.892
C09886=1171.291,76.740,-50.512,-179.258,6.169,148.893
C09887=1171.296,76.490,-50.495,-179.260,6.168,148.893
C09888=1171.301,76.241,-50.479,-179.263,6.166,148.894
C09889=1171.306,75.992,-50.461,-179.266,6.166,148.894
C09890=1171.311,75.743,-50.444,-179.269,6.164,148.895
C09891=1171.316,75.493,-50.427,-179.271,6.163,148.895
C09892=1171.320,75.243,-50.410,-179.274,6.162,148.896
C09893=1171.326,74.995,-50.393,-179.276,6.161,148.896
C09894=1171.330,74.745,-50.376,-179.279,6.161,148.897
C09895=1171.336,74.496,-50.359,-179.282,6.159,148.898
C09896=1171.340,74.246,-50.342,-179.284,6.158,148.898
C09897=1171.346,73.997,-50.325,-179.287,6.157,148.899
C09898=1171.350,73.748,-50.309,-179.289,6.156,148.899
C09899=1171.355,73.498,-50.291,-179.292,6.154,148.900
C09900=1171.360,73.249,-50.274,-179.294,6.154,148.900
C09901=1171.365,72.999,-50.257,-179.298,6.152,148.901
C09902=1171.370,72.750,-50.240,-179.300,6.151,148.901
C09903=1171.375,72.500,-50.223,-179.303,6.150,148.902
C09904=1171.380,72.251,-50.206,-179.305,6.149,148.902
C09905=1171.385,72.001,-50.189,-179.308,6.148,148.903
C09906=1171.390,71.752,-50.173,-179.311,6.147,148.903
C09907=1171.395,71.503,-50.156,-179.313,6.146,148.904
C09908=1171.399,71.254,-50.138,-179.316,6.145,148.904
C09909=1171.405,71.005,-50.122,-179.318,6.144,148.905
C09910=1171.410,70.755,-50.105,-179.321,6.142,148.906
C09911=1171.414,70.506,-50.088,-179.323,6.142,148.906
C09912=1171.419,70.256,-50.071,-179.327,6.140,148.907
C09913=1171.425,70.007,-50.054,-179.329,6.139,148.907
C09914=1171.429,69.758,-50.038,-179.332,6.138,148.908
C09915=1171.434,69.508,-50.020,-179.334,6.137,148.908
C09916=1171.439,69.259,-50.004,-179.337,6.137,148.909
C09917=1171.444,69.010,-49.987,-179.340,6.135,148.909
C09918=1171.449,68.760,-49.970,-179.342,6.134,148.910
C09919=1171.454,68.511,-49.954,-179.345,6.133,148.910
C09920=1171.459,68.262,-49.937,-179.348,6.132,148.911
C09921=1171.464,68.011,-49.921,-179.350,6.131,148.911
C09922=1171.469,67.762,-49.904,-179.353,6.130,148.912
C09923=1171.474,67.513,-49.888,-179.356,6.128,148.913
C09924=1171.479,67.263,-49.870,-179.358,6.128,148.913
C09925=1171.484,67.014,-49.854,-179.360,6.127,148.914
C09926=1171.488,66.765,-49.837,-179.363,6.125,148.914
C09927=1171.494,66.515,-49.820,-179.366,6.125,148.915
C09928=1171.499,66.266,-49.804,-179.369,6.123,148.915
C09929=1171.503,66.017,-49.787,-179.371,6.123,148.916
C09930=1171.508,65.767,-49.771,-179.373,6.122,148.916
C09931=1171.514,65.518,-49.754,-179.377,6.120,148.917
C09932=1171.518,65.268,-49.738,-179.379,6.119,148.917
C09933=1171.523,65.019,-49.721,-179.382,6.118,148.918
C09934=1171.528,64.770,-49.705,-179.384,6.117,148.918
C09935=1171.533,64.520,-49.687,-179.387,6.116,148.919
C09936=1171.539,64.271,-49.672,-179.389,6.115,148.920
C09937=1171.543,64.021,-49.655,-179.392,6.115,148.920
C09938=1171.547,63.772,-49.639,-179.395,6.113,148.921
C09939=1171.553,63.523,-49.622,-179.397,6.112,148.921
C09940=1171.558,63.273,-49.605,-179.400,6.111,148.922
C09941=1171.563,63.024,-49.589,-179.403,6.110,148.922
C09942=1171.568,62.774,-49.573,-179.405,6.109,148.923
C09943=1171.573,62.525,-49.556,-179.408,6.108,148.923
C09944=1171.577,62.275,-49.540,-179.410,6.107,148.924
C09945=1171.583,62.025,-49.523,-179.413,6.107,148.925
C09946=1171.588,61.777,-49.507,-179.416,6.105,148.925
C09947=1171.592,61.527,-49.490,-179.418,6.104,148.926
C09948=1171.598,61.278,-49.475,-179.421,6.103,148.926
C09949=1171.602,61.028,-49.458,-179.424,6.102,148.927
C09950=1171.607,60.780,-49.442,-179.426,6.101,148.927
C09951=1171.613,60.529,-49.425,-179.429,6.100,148.928
C09952=1171.618,60.280,-49.409,-179.431,6.099,148.928
C09953=1171.622,60.031,-49.392,-179.434,6.098,148.929
C09954=1171.628,59.781,-49.377,-179.437,6.097,148.929
C09955=1171.632,59.532,-49.360,-179.439,6.096,148.930
C09956=1171.638,59.283,-49.344,-179.442,6.095,148.931
C09957=1171.642,59.033,-49.328,-179.445,6.094,148.931
C09958=1171.647,58.784,-49.311,-179.447,6.093,148.932
C09959=1171.652,58.534,-49.295,-179.450,6.092,148.932
C09960=1171.656,58.285,-49.279,-179.452,6.091,148.933
C09961=1171.663,58.035,-49.263,-179.455,6.090,148.933
C09962=1171.668,57.786,-49.246,-179.457,6.089,148.934
C09963=1171.672,57.536,-49.230,-179.460,6.088,148.934
C09964=1171.677,57.287,-49.214,-179.463,6.087,148.935
C09965=1171.682,57.037,-49.198,-179.465,6.086,148.936
C09966=1171.687,56.788,-49.182,-179.468,6.085,148.936
C09967=1171.692,56.538,-49.166,-179.471,6.084,148.937
C09968=1171.697,56.290,-49.149,-179.473,6.083,148.937
C09969=1171.702,56.039,-49.134,-179.476,6.083,148.938
C09970=1171.707,55.791,-49.117,-179.479,6.081,148.938
C09971=1171.712,55.541,-49.101,-179.481,6.081,148.939
C09972=1171.717,55.292,-49.085,-179.484,6.080,148.940
C09973=1171.722,55.042,-49.069,-179.486,6.078,148.940
C09974=1171.727,54.793,-49.053,-179.489,6.078,148.941
C09975=1171.732,54.524,-49.036,-179.492,6.076,148.941
C09976=1171.737,54.255,-49.018,-179.494,6.076,148.942
C09977=1171.743,53.987,-49.001,-179.498,6.074,148.942
C09978=1171.748,53.718,-48.984,-179.500,6.073,148.943
C09979=1171.754,53.469,-48.968,-179.503,6.072,148.944
C09980=1171.758,53.219,-48.952,-179.506,6.072,148.944
C09981=1171.763,52.971,-48.936,-179.508,6.071,148.945
C09982=1171.768,52.720,-48.920,-179.511,6.069,148.945
C09983=1171.774,52.471,-48.904,-179.513,6.069,148.946
C09984=1171.779,52.222,-48.888,-179.516,6.068,148.946
C09985=1171.783,51.972,-48.872,-179.519,6.066,148.947
C09986=1171.788,51.723,-48.857,-179.521,6.066,148.948
C09987=1171.793,51.474,-48.840,-179.523,6.065,148.948
C09988=1171.798,51.224,-48.825,-179.527,6.064,148.949
C09989=1171.803,50.975,-48.809,-179.529,6.063,148.949
C09990=1171.808,50.725,-48.792,-179.531,6.062,148.950
C09991=1171.813,50.476,-48.777,-179.534,6.061,148.950
C09992=1171.818,50.226,-48.761,-179.537,6.060,148.951
C09993=1171.823,49.976,-48.745,-179.539,6.059,148.951
C09994=1171.828,49.728,-48.730,-179.542,6.059,148.952
C09995=1171.832,49.478,-48.714,-179.545,6.057,148.953
C09996=1171.838,49.228,-48.698,-179.547,6.057,148.953
//INST
///DATE 2021/06/25 14:30
///ATTR SC,RW,RJ
////FRAME ROBOT
///GROUP1 RB1
NOP
MOVL C00000 V=800.0 PL=0
MOVL C00001 V=800.0 PL=0
MOVL C00002 V=800.0 PL=0
MOVL C00003 V=800.0 PL=0
MOVL C00004 V=800.0 PL=0
MOVL C00005 V=800.0 PL=0
MOVL C00006 V=800.0 PL=0
MOVL C00007 V=800.0 PL=0
MOVL C00008 V=800.0 PL=0
MOVL C00009 V=800.0 PL=0
MOVL C00010 V=800.0 PL=0
MOVL C00011 V=800.0 PL=0
MOVL C00012 V=800.0 PL=0
MOVL C00013 V=800.0 PL=0
MOVL C00014 V=800.0 PL=0
MOVL C00015 V=800.0 PL=0
MOVL C00016 V=800.0 PL=0
MOVL C00017 V=800.0 PL=0
MOVL C00018 V=800.0 PL=0
MOVL C00019 V=800.0 PL=0
MOVL C00020 V=800.0 PL=0
MOVL C00021 V=800.0 PL=0
MOVL C00022 V=800.0 PL=0
MOVL C00023 V=800.0 PL=0
MOVL C00024 V=800.0 PL=0
MOVL C00025 V=800.0 PL=0
MOVL C00026 V=800.0 PL=0
MOVL C00027 V=800.0 PL=0
MOVL C00028 V=800.0 PL=0
MOVL C00029 V=800.0 PL=0
MOVL C00030 V=800.0 PL=0
MOVL C00031 V=800.0 PL=0
MOVL C00032 V=800.0 PL=0
MOVL C00033 V=800.0 PL=0
MOVL C00034 V=800.0 PL=0
MOVL C00035 V=800.0 PL=0
MOVL C00036 V=800.0 PL=0
MOVL C00037 V=800.0 PL=0
MOVL C00038 V=800.0 PL=0
MOVL C00039 V=800.0 PL=0
MOVL C00040 V=800.0 PL=0
MOVL C00041 V=800.0 PL=0
MOVL C00042 V=800.0 PL=0
MOVL C00043 V=800.0 PL=0
MOVL C00044 V=800.0 PL=0
MOVL C00045 V=800.0 PL=0
MOVL C00046 V=800.0 PL=0
MOVL C00047 V=800.0 PL=0
MOVL C00048 V=800.0 PL=0
MOVL C00049 V=800.0 PL=0
MOVL C00050 V=800.0 PL=0
MOVL C00051 V=800.0 PL=0
MOVL C00052 V=800.0 PL=0
MOVL C00053 V=800.0 PL=0
MOVL C00054 V=800.0 PL=0
MOVL C00055 V=800.0 PL=0
MOVL C00056 V=800.0 PL=0
MOVL C00057 V=800.0 PL=0
MOVL C00058 V=800.0 PL=0
MOVL C00059 V=800.0 PL=0
MOVL C00060 V=800.0 PL=0
MOVL C00061 V=800.0 PL=0
MOVL C00062 V=800.0 PL=0
MOVL C00063 V=800.0 PL=0
MOVL C00064 V=800.0 PL=0
MOVL C00065 V=800.0 PL=0
MOVL C00066 V=800.0 PL=0
MOVL C00067 V=800.0 PL=0
MOVL C00068 V=800.0 PL=0
MOVL C00069 V=800.0 PL=0
MOVL C00070 V=800.0 PL=0
MOVL C00071 V=800.0 PL=0
MOVL C00072 V=800.0 PL=0
MOVL C00073 V=800.0 PL=0
MOVL C00074 V=800.0 PL=0
MOVL C00075 V=800.0 PL=0
MOVL C00076 V=800.0 PL=0
MOVL C00077 V=800.0 PL=0
MOVL C00078 V=800.0 PL=0
MOVL C00079 V=800.0 PL=0
MOVL C00080 V=800.0 PL=0
MOVL C00081 V=800.0 PL=0
MOVL C00082 V=800.0 PL=0
MOVL C00083 V=800.0 PL=0
MOVL C00084 V=800.0 PL=0
MOVL C00085 V=800.0 PL=0
MOVL C00086 V=800.0 PL=0
MOVL C00087 V=800.0 PL=0
MOVL C00088 V=800.0 PL=0
MOVL C00089 V=800.0 PL=0
MOVL C00090 V=800.0 PL=0
MOVL C00091 V=800.0 PL=0
MOVL C00092 V=800.0 PL=0
MOVL C00093 V=800.0 PL=0
MOVL C00094 V=800.0 PL=0
MOVL C00095 V=800.0 PL=0
MOVL C00096 V=800.0 PL=0
MOVL C00097 V=800.0 PL=0
MOVL C00098 V=800.0 PL=0
MOVL C00099 V=800.0 PL=0
MOVL C00100 V=800.0 PL=0
MOVL C00101 V=800.0 PL=0
MOVL C00102 V=800.0 PL=0
MOVL C00103 V=800.0 PL=0
MOVL C00104 V=800.0 PL=0
MOVL C00105 V=800.0 PL=0
MOVL C00106 V=800.0 PL=0
MOVL C00107 V=800.0 PL=0
MOVL C00108 V=800.0 PL=0
MOVL C00109 V=800.0 PL=0
MOVL C00110 V=800.0 PL=0
MOVL C00111 V=800.0 PL=0
MOVL C00112 V=800.0 PL=0
MOVL C00113 V=800.0 PL=0
MOVL C00114 V=800.0 PL=0
MOVL C00115 V=800.0 PL=0
MOVL C00116 V=800.0 PL=0
MOVL C00117 V=800.0 PL=0
MOVL C00118 V=800.0 PL=0
MOVL C00119 V=800.0 PL=0
MOVL C00120 V=800.0 PL=0
MOVL C00121 V=800.0 PL=0
MOVL C00122 V=800.0 PL=0
MOVL C00123 V=800.0 PL=0
MOVL C00124 V=800.0 PL=0
MOVL C00125 V=800.0 PL=0
MOVL C00126 V=800.0 PL=0
MOVL C00127 V=800.0 PL=0
MOVL C00128 V=800.0 PL=0
MOVL C00129 V=800.0 PL=0
MOVL C00130 V=800.0 PL=0
MOVL C00131 V=800.0 PL=0
MOVL C00132 V=800.0 PL=0
MOVL C00133 V=800.0 PL=0
MOVL C00134 V=800.0 PL=0
MOVL C00135 V=800.0 PL=0
MOVL C00136 V=800.0 PL=0
MOVL C00137 V=800.0 PL=0
MOVL C00138 V=800.0 PL=0
MOVL C00139 V=800.0 PL=0
MOVL C00140 V=800.0 PL=0
MOVL C00141 V=800.0 PL=0
MOVL C00142 V=800.0 PL=0
MOVL C00143 V=800.0 PL=0
MOVL C00144 V=800.0 PL=0
MOVL C00145 V=800.0 PL=0
MOVL C00146 V=800.0 PL=0
MOVL C00147 V=800.0 PL=0
MOVL C00148 V=800.0 PL=0
MOVL C00149 V=800.0 PL=0
MOVL C00150 V=800.0 PL=0
MOVL C00151 V=800.0 PL=0
MOVL C00152 V=800.0 PL=0
MOVL C00153 V=800.0 PL=0
MOVL C00154 V=800.0 PL=0
MOVL C00155 V=800.0 PL=0
MOVL C00156 V=800.0 PL=0
MOVL C00157 V=800.0 PL=0
MOVL C00158 V=800.0 PL=0
MOVL C00159 V=800.0 PL=0
MOVL C00160 V=800.0 PL=0
MOVL C00161 V=800.0 PL=0
MOVL C00162 V=800.0 PL=0
MOVL C00163 V=800.0 PL=0
MOVL C00164 V=800.0 PL=0
MOVL C00165 V=800.0 PL=0
MOVL C00166 V=800.0 PL=0
MOVL C00167 V=800.0 PL=0
MOVL C00168 V=800.0 PL=0
MOVL C00169 V=800.0 PL=0
MOVL C00170 V=800.0 PL=0
MOVL C00171 V=800.0 PL=0
MOVL C00172 V=800.0 PL=0
MOVL C00173 V=800.0 PL=0
MOVL C00174 V=800.0 PL=0
MOVL C00175 V=800.0 PL=0
MOVL C00176 V=800.0 PL=0
MOVL C00177 V=800.0 PL=0
MOVL C00178 V=800.0 PL=0
MOVL C00179 V=800.0 PL=0
MOVL C00180 V=800.0 PL=0
MOVL C00181 V=800.0 PL=0
MOVL C00182 V=800.0 PL=0
MOVL C00183 V=800.0 PL=0
MOVL C00184 V=800.0 PL=0
MOVL C00185 V=800.0 PL=0
MOVL C00186 V=800.0 PL=0
MOVL C00187 V=800.0 PL=0
MOVL C00188 V=800.0 PL=0
MOVL C00189 V=800.0 PL=0
MOVL C00190 V=800.0 PL=0
MOVL C00191 V=800.0 PL=0
MOVL C00192 V=800.0 PL=0
MOVL C00193 V=800.0 PL=0
MOVL C00194 V=800.0 PL=0
MOVL C00195 V=800.0 PL=0
MOVL C00196 V=800.0 PL=0
MOVL C00197 V=800.0 PL=0
MOVL C00198 V=800.0 PL=0
MOVL C00199 V=800.0 PL=0
MOVL C00200 V=800.0 PL=0
MOVL C00201 V=800.0 PL=0
MOVL C00202 V=800.0 PL=0
MOVL C00203 V=800.0 PL=0
MOVL C00204 V=800.0 PL=0
MOVL C00205 V=800.0 PL=0
MOVL C00206 V=800.0 PL=0
MOVL C00207 V=800.0 PL=0
MOVL C00208 V=800.0 PL=0
MOVL C00209 V=800.0 PL=0
MOVL C00210 V=800.0 PL=0
MOVL C00211 V=800.0 PL=0
MOVL C00212 V=800.0 PL=0
MOVL C00213 V=800.0 PL=0
MOVL C00214 V=800.0 PL=0
MOVL C00215 V=800.0 PL=0
MOVL C00216 V=800.0 PL=0
MOVL C00217 V=800.0 PL=0
MOVL C00218 V=800.0 PL=0
MOVL C00219 V=800.0 PL=0
MOVL C00220 V=800.0 PL=0
MOVL C00221 V=800.0 PL=0
MOVL C00222 V=800.0 PL=0
MOVL C00223 V=800.0 PL=0
MOVL C00224 V=800.0 PL=0
MOVL C00225 V=800.0 PL=0
MOVL C00226 V=800.0 PL=0
MOVL C00227 V=800.0 PL=0
MOVL C00228 V=800.0 PL=0
MOVL C00229 V=800.0 PL=0
MOVL C00230 V=800.0 PL=0
MOVL C00231 V=800.0 PL=0
MOVL C00232 V=800.0 PL=0
MOVL C00233 V=800.0 PL=0
MOVL C00234 V=800.0 PL=0
MOVL C00235 V=800.0 PL=0
MOVL C00236 V=800.0 PL=0
MOVL C00237 V=800.0 PL=0
MOVL C00238 V=800.0 PL=0
MOVL C00239 V=800.0 PL=0
MOVL C00240 V=800.0 PL=0
MOVL C00241 V=800.0 PL=0
MOVL C00242 V=800.0 PL=0
MOVL C00243 V=800.0 PL=0
MOVL C00244 V=800.0 PL=0
MOVL C00245 V=800.0 PL=0
MOVL C00246 V=800.0 PL=0
MOVL C00247 V=800.0 PL=0
MOVL C00248 V=800.0 PL=0
MOVL C00249 V=800.0 PL=0
MOVL C00250 V=800.0 PL=0
MOVL C00251 V=800.0 PL=0
MOVL C00252 V=800.0 PL=0
MOVL C00253 V=800.0 PL=0
MOVL C00254 V=800.0 PL=0
MOVL C00255 V=800.0 PL=0
MOVL C00256 V=800.0 PL=0
MOVL C00257 V=800.0 PL=0
MOVL C00258 V=800.0 PL=0
MOVL C00259 V=800.0 PL=0
MOVL C00260 V=800.0 PL=0
MOVL C00261 V=800.0 PL=0
MOVL C00262 V=800.0 PL=0
MOVL C00263 V=800.0 PL=0
MOVL C00264 V=800.0 PL=0
MOVL C00265 V=800.0 PL=0
MOVL C00266 V=800.0 PL=0
MOVL C00267 V=800.0 PL=0
MOVL C00268 V=800.0 PL=0
MOVL C00269 V=800.0 PL=0
MOVL C00270 V=800.0 PL=0
MOVL C00271 V=800.0 PL=0
MOVL C00272 V=800.0 PL=0
MOVL C00273 V=800.0 PL=0
MOVL C00274 V=800.0 PL=0
MOVL C00275 V=800.0 PL=0
MOVL C00276 V=800.0 PL=0
MOVL C00277 V=800.0 PL=0
MOVL C00278 V=800.0 PL=0
MOVL C00279 V=800.0 PL=0
MOVL C00280 V=800.0 PL=0
MOVL C00281 V=800.0 PL=0
MOVL C00282 V=800.0 PL=0
MOVL C00283 V=800.0 PL=0
MOVL C00284 V=800.0 PL=0
MOVL C00285 V=800.0 PL=0
MOVL C00286 V=800.0 PL=0
MOVL C00287 V=800.0 PL=0
MOVL C00288 V=800.0 PL=0
MOVL C00289 V=800.0 PL=0
MOVL C00290 V=800.0 PL=0
MOVL C00291 V=800.0 PL=0
MOVL C00292 V=800.0 PL=0
MOVL C00293 V=800.0 PL=0
MOVL C00294 V=800.0 PL=0
MOVL C00295 V=800.0 PL=0
MOVL C00296 V=800.0 PL=0
MOVL C00297 V=800.0 PL=0
MOVL C00298 V=800.0 PL=0
MOVL C00299 V=800.0 PL=0
MOVL C00300 V=800.0 PL=0
MOVL C00301 V=800.0 PL=0
MOVL C00302 V=800.0 PL=0
MOVL C00303 V=800.0 PL=0
MOVL C00304 V=800.0 PL=0
MOVL C00305 V=800.0 PL=0
MOVL C00306 V=800.0 PL=0
MOVL C00307 V=800.0 PL=0
MOVL C00308 V=800.0 PL=0
MOVL C00309 V=800.0 PL=0
MOVL C00310 V=800.0 PL=0
MOVL C00311 V=800.0 PL=0
MOVL C00312 V=800.0 PL=0
MOVL C00313 V=800.0 PL=0
MOVL C00314 V=800.0 PL=0
MOVL C00315 V=800.0 PL=0
MOVL C00316 V=800.0 PL=0
MOVL C00317 V=800.0 PL=0
MOVL C00318 V=800.0 PL=0
MOVL C00319 V=800.0 PL=0
MOVL C00320 V=800.0 PL=0
MOVL C00321 V=800.0 PL=0
MOVL C00322 V=800.0 PL=0
MOVL C00323 V=800.0 PL=0
MOVL C00324 V=800.0 PL=0
MOVL C00325 V=800.0 PL=0
MOVL C00326 V=800.0 PL=0
MOVL C00327 V=800.0 PL=0
MOVL C00328 V=800.0 PL=0
MOVL C00329 V=800.0 PL=0
MOVL C00330 V=800.0 PL=0
MOVL C00331 V=800.0 PL=0
MOVL C00332 V=800.0 PL=0
MOVL C00333 V=800.0 PL=0
MOVL C00334 V=800.0 PL=0
MOVL C00335 V=800.0 PL=0
MOVL C00336 V=800.0 PL=0
MOVL C00337 V=800.0 PL=0
MOVL C00338 V=800.0 PL=0
MOVL C00339 V=800.0 PL=0
MOVL C00340 V=800.0 PL=0
MOVL C00341 V=800.0 PL=0
MOVL C00342 V=800.0 PL=0
MOVL C00343 V=800.0 PL=0
MOVL C00344 V=800.0 PL=0
MOVL C00345 V=800.0 PL=0
MOVL C00346 V=800.0 PL=0
MOVL C00347 V=800.0 PL=0
MOVL C00348 V=800.0 PL=0
MOVL C00349 V=800.0 PL=0
MOVL C00350 V=800.0 PL=0
MOVL C00351 V=800.0 PL=0
MOVL C00352 V=800.0 PL=0
MOVL C00353 V=800.0 PL=0
MOVL C00354 V=800.0 PL=0
MOVL C00355 V=800.0 PL=0
MOVL C00356 V=800.0 PL=0
MOVL C00357 V=800.0 PL=0
MOVL C00358 V=800.0 PL=0
MOVL C00359 V=800.0 PL=0
MOVL C00360 V=800.0 PL=0
MOVL C00361 V=800.0 PL=0
MOVL C00362 V=800.0 PL=0
MOVL C00363 V=800.0 PL=0
MOVL C00364 V=800.0 PL=0
MOVL C00365 V=800.0 PL=0
MOVL C00366 V=800.0 PL=0
MOVL C00367 V=800.0 PL=0
MOVL C00368 V=800.0 PL=0
MOVL C00369 V=800.0 PL=0
MOVL C00370 V=800.0 PL=0
MOVL C00371 V=800.0 PL=0
MOVL C00372 V=800.0 PL=0
MOVL C00373 V=800.0 PL=0
MOVL C00374 V=800.0 PL=0
MOVL C00375 V=800.0 PL=0
MOVL C00376 V=800.0 PL=0
MOVL C00377 V=800.0 PL=0
MOVL C00378 V=800.0 PL=0
MOVL C00379 V=800.0 PL=0
MOVL C00380 V=800.0 PL=0
MOVL C00381 V=800.0 PL=0
MOVL C00382 V=800.0 PL=0
MOVL C00383 V=800.0 PL=0
MOVL C00384 V=800.0 PL=0
MOVL C00385 V=800.0 PL=0
MOVL C00386 V=800.0 PL=0
MOVL C00387 V=800.0 PL=0
MOVL C00388 V=800.0 PL=0
MOVL C00389 V=800.0 PL=0
MOVL C00390 V=800.0 PL=0
MOVL C00391 V=800.0 PL=0
MOVL C00392 V=800.0 PL=0
MOVL C00393 V=800.0 PL=0
MOVL C00394 V=800.0 PL=0
MOVL C00395 V=800.0 PL=0
MOVL C00396 V=800.0 PL=0
MOVL C00397 V=800.0 PL=0
MOVL C00398 V=800.0 PL=0
MOVL C00399 V=800.0 PL=0
MOVL C00400 V=800.0 PL=0
MOVL C00401 V=800.0 PL=0
MOVL C00402 V=800.0 PL=0
MOVL C00403 V=800.0 PL=0
MOVL C00404 V=800.0 PL=0
MOVL C00405 V=800.0 PL=0
MOVL C00406 V=800.0 PL=0
MOVL C00407 V=800.0 PL=0
MOVL C00408 V=800.0 PL=0
MOVL C00409 V=800.0 PL=0
MOVL C00410 V=800.0 PL=0
MOVL C00411 V=800.0 PL=0
MOVL C00412 V=800.0 PL=0
MOVL C00413 V=800.0 PL=0
MOVL C00414 V=800.0 PL=0
MOVL C00415 V=800.0 PL=0
MOVL C00416 V=800.0 PL=0
MOVL C00417 V=800.0 PL=0
MOVL C00418 V=800.0 PL=0
MOVL C00419 V=800.0 PL=0
MOVL C00420 V=800.0 PL=0
MOVL C00421 V=800.0 PL=0
MOVL C00422 V=800.0 PL=0
MOVL C00423 V=800.0 PL=0
MOVL C00424 V=800.0 PL=0
MOVL C00425 V=800.0 PL=0
MOVL C00426 V=800.0 PL=0
MOVL C00427 V=800.0 PL=0
MOVL C00428 V=800.0 PL=0
MOVL C00429 V=800.0 PL=0
MOVL C00430 V=800.0 PL=0
MOVL C00431 V=800.0 PL=0
MOVL C00432 V=800.0 PL=0
MOVL C00433 V=800.0 PL=0
MOVL C00434 V=800.0 PL=0
MOVL C00435 V=800.0 PL=0
MOVL C00436 V=800.0 PL=0
MOVL C00437 V=800.0 PL=0
MOVL C00438 V=800.0 PL=0
MOVL C00439 V=800.0 PL=0
MOVL C00440 V=800.0 PL=0
MOVL C00441 V=800.0 PL=0
MOVL C00442 V=800.0 PL=0
MOVL C00443 V=800.0 PL=0
MOVL C00444 V=800.0 PL=0
MOVL C00445 V=800.0 PL=0
MOVL C00446 V=800.0 PL=0
MOVL C00447 V=800.0 PL=0
MOVL C00448 V=800.0 PL=0
MOVL C00449 V=800.0 PL=0
MOVL C00450 V=800.0 PL=0
MOVL C00451 V=800.0 PL=0
MOVL C00452 V=800.0 PL=0
MOVL C00453 V=800.0 PL=0
MOVL C00454 V=800.0 PL=0
MOVL C00455 V=800.0 PL=0
MOVL C00456 V=800.0 PL=0
MOVL C00457 V=800.0 PL=0
MOVL C00458 V=800.0 PL=0
MOVL C00459 V=800.0 PL=0
MOVL C00460 V=800.0 PL=0
MOVL C00461 V=800.0 PL=0
MOVL C00462 V=800.0 PL=0
MOVL C00463 V=800.0 PL=0
MOVL C00464 V=800.0 PL=0
MOVL C00465 V=800.0 PL=0
MOVL C00466 V=800.0 PL=0
MOVL C00467 V=800.0 PL=0
MOVL C00468 V=800.0 PL=0
MOVL C00469 V=800.0 PL=0
MOVL C00470 V=800.0 PL=0
MOVL C00471 V=800.0 PL=0
MOVL C00472 V=800.0 PL=0
MOVL C00473 V=800.0 PL=0
MOVL C00474 V=800.0 PL=0
MOVL C00475 V=800.0 PL=0
MOVL C00476 V=800.0 PL=0
MOVL C00477 V=800.0 PL=0
MOVL C00478 V=800.0 PL=0
MOVL C00479 V=800.0 PL=0
MOVL C00480 V=800.0 PL=0
MOVL C00481 V=800.0 PL=0
MOVL C00482 V=800.0 PL=0
MOVL C00483 V=800.0 PL=0
MOVL C00484 V=800.0 PL=0
MOVL C00485 V=800.0 PL=0
MOVL C00486 V=800.0 PL=0
MOVL C00487 V=800.0 PL=0
MOVL C00488 V=800.0 PL=0
MOVL C00489 V=800.0 PL=0
MOVL C00490 V=800.0 PL=0
MOVL C00491 V=800.0 PL=0
MOVL C00492 V=800.0 PL=0
MOVL C00493 V=800.0 PL=0
MOVL C00494 V=800.0 PL=0
MOVL C00495 V=800.0 PL=0
MOVL C00496 V=800.0 PL=0
MOVL C00497 V=800.0 PL=0
MOVL C00498 V=800.0 PL=0
MOVL C00499 V=800.0 PL=0
MOVL C00500 V=800.0 PL=0
MOVL C00501 V=800.0 PL=0
MOVL C00502 V=800.0 PL=0
MOVL C00503 V=800.0 PL=0
MOVL C00504 V=800.0 PL=0
MOVL C00505 V=800.0 PL=0
MOVL C00506 V=800.0 PL=0
MOVL C00507 V=800.0 PL=0
MOVL C00508 V=800.0 PL=0
MOVL C00509 V=800.0 PL=0
MOVL C00510 V=800.0 PL=0
MOVL C00511 V=800.0 PL=0
MOVL C00512 V=800.0 PL=0
MOVL C00513 V=800.0 PL=0
MOVL C00514 V=800.0 PL=0
MOVL C00515 V=800.0 PL=0
MOVL C00516 V=800.0 PL=0
MOVL C00517 V=800.0 PL=0
MOVL C00518 V=800.0 PL=0
MOVL C00519 V=800.0 PL=0
MOVL C00520 V=800.0 PL=0
MOVL C00521 V=800.0 PL=0
MOVL C00522 V=800.0 PL=0
MOVL C00523 V=800.0 PL=0
MOVL C00524 V=800.0 PL=0
MOVL C00525 V=800.0 PL=0
MOVL C00526 V=800.0 PL=0
MOVL C00527 V=800.0 PL=0
MOVL C00528 V=800.0 PL=0
MOVL C00529 V=800.0 PL=0
MOVL C00530 V=800.0 PL=0
MOVL C00531 V=800.0 PL=0
MOVL C00532 V=800.0 PL=0
MOVL C00533 V=800.0 PL=0
MOVL C00534 V=800.0 PL=0
MOVL C00535 V=800.0 PL=0
MOVL C00536 V=800.0 PL=0
MOVL C00537 V=800.0 PL=0
MOVL C00538 V=800.0 PL=0
MOVL C00539 V=800.0 PL=0
MOVL C00540 V=800.0 PL=0
MOVL C00541 V=800.0 PL=0
MOVL C00542 V=800.0 PL=0
MOVL C00543 V=800.0 PL=0
MOVL C00544 V=800.0 PL=0
MOVL C00545 V=800.0 PL=0
MOVL C00546 V=800.0 PL=0
MOVL C00547 V=800.0 PL=0
MOVL C00548 V=800.0 PL=0
MOVL C00549 V=800.0 PL=0
MOVL C00550 V=800.0 PL=0
MOVL C00551 V=800.0 PL=0
MOVL C00552 V=800.0 PL=0
MOVL C00553 V=800.0 PL=0
MOVL C00554 V=800.0 PL=0
MOVL C00555 V=800.0 PL=0
MOVL C00556 V=800.0 PL=0
MOVL C00557 V=800.0 PL=0
MOVL C00558 V=800.0 PL=0
MOVL C00559 V=800.0 PL=0
MOVL C00560 V=800.0 PL=0
MOVL C00561 V=800.0 PL=0
MOVL C00562 V=800.0 PL=0
MOVL C00563 V=800.0 PL=0
MOVL C00564 V=800.0 PL=0
MOVL C00565 V=800.0 PL=0
MOVL C00566 V=800.0 PL=0
MOVL C00567 V=800.0 PL=0
MOVL C00568 V=800.0 PL=0
MOVL C00569 V=800.0 PL=0
MOVL C00570 V=800.0 PL=0
MOVL C00571 V=800.0 PL=0
MOVL C00572 V=800.0 PL=0
MOVL C00573 V=800.0 PL=0
MOVL C00574 V=800.0 PL=0
MOVL C00575 V=800.0 PL=0
MOVL C00576 V=800.0 PL=0
MOVL C00577 V=800.0 PL=0
MOVL C00578 V=800.0 PL=0
MOVL C00579 V=800.0 PL=0
MOVL C00580 V=800.0 PL=0
MOVL C00581 V=800.0 PL=0
MOVL C00582 V=800.0 PL=0
MOVL C00583 V=800.0 PL=0
MOVL C00584 V=800.0 PL=0
MOVL C00585 V=800.0 PL=0
MOVL C00586 V=800.0 PL=0
MOVL C00587 V=800.0 PL=0
MOVL C00588 V=800.0 PL=0
MOVL C00589 V=800.0 PL=0
MOVL C00590 V=800.0 PL=0
MOVL C00591 V=800.0 PL=0
MOVL C00592 V=800.0 PL=0
MOVL C00593 V=800.0 PL=0
MOVL C00594 V=800.0 PL=0
MOVL C00595 V=800.0 PL=0
MOVL C00596 V=800.0 PL=0
MOVL C00597 V=800.0 PL=0
MOVL C00598 V=800.0 PL=0
MOVL C00599 V=800.0 PL=0
MOVL C00600 V=800.0 PL=0
MOVL C00601 V=800.0 PL=0
MOVL C00602 V=800.0 PL=0
MOVL C00603 V=800.0 PL=0
MOVL C00604 V=800.0 PL=0
MOVL C00605 V=800.0 PL=0
MOVL C00606 V=800.0 PL=0
MOVL C00607 V=800.0 PL=0
MOVL C00608 V=800.0 PL=0
MOVL C00609 V=800.0 PL=0
MOVL C00610 V=800.0 PL=0
MOVL C00611 V=800.0 PL=0
MOVL C00612 V=800.0 PL=0
MOVL C00613 V=800.0 PL=0
MOVL C00614 V=800.0 PL=0
MOVL C00615 V=800.0 PL=0
MOVL C00616 V=800.0 PL=0
MOVL C00617 V=800.0 PL=0
MOVL C00618 V=800.0 PL=0
MOVL C00619 V=800.0 PL=0
MOVL C00620 V=800.0 PL=0
MOVL C00621 V=800.0 PL=0
MOVL C00622 V=800.0 PL=0
MOVL C00623 V=800.0 PL=0
MOVL C00624 V=800.0 PL=0
MOVL C00625 V=800.0 PL=0
MOVL C00626 V=800.0 PL=0
MOVL C00627 V=800.0 PL=0
MOVL C00628 V=800.0 PL=0
MOVL C00629 V=800.0 PL=0
MOVL C00630 V=800.0 PL=0
MOVL C00631 V=800.0 PL=0
MOVL C00632 V=800.0 PL=0
MOVL C00633 V=800.0 PL=0
MOVL C00634 V=800.0 PL=0
MOVL C00635 V=800.0 PL=0
MOVL C00636 V=800.0 PL=0
MOVL C00637 V=800.0 PL=0
MOVL C00638 V=800.0 PL=0
MOVL C00639 V=800.0 PL=0
MOVL C00640 V=800.0 PL=0
MOVL C00641 V=800.0 PL=0
MOVL C00642 V=800.0 PL=0
MOVL C00643 V=800.0 PL=0
MOVL C00644 V=800.0 PL=0
MOVL C00645 V=800.0 PL=0
MOVL C00646 V=800.0 PL=0
MOVL C00647 V=800.0 PL=0
MOVL C00648 V=800.0 PL=0
MOVL C00649 V=800.0 PL=0
MOVL C00650 V=800.0 PL=0
MOVL C00651 V=800.0 PL=0
MOVL C00652 V=800.0 PL=0
MOVL C00653 V=800.0 PL=0
MOVL C00654 V=800.0 PL=0
MOVL C00655 V=800.0 PL=0
MOVL C00656 V=800.0 PL=0
MOVL C00657 V=800.0 PL=0
MOVL C00658 V=800.0 PL=0
MOVL C00659 V=800.0 PL=0
MOVL C00660 V=800.0 PL=0
MOVL C00661 V=800.0 PL=0
MOVL C00662 V=800.0 PL=0
MOVL C00663 V=800.0 PL=0
MOVL C00664 V=800.0 PL=0
MOVL C00665 V=800.0 PL=0
MOVL C00666 V=800.0 PL=0
MOVL C00667 V=800.0 PL=0
MOVL C00668 V=800.0 PL=0
MOVL C00669 V=800.0 PL=0
MOVL C00670 V=800.0 PL=0
MOVL C00671 V=800.0 PL=0
MOVL C00672 V=800.0 PL=0
MOVL C00673 V=800.0 PL=0
MOVL C00674 V=800.0 PL=0
MOVL C00675 V=800.0 PL=0
MOVL C00676 V=800.0 PL=0
MOVL C00677 V=800.0 PL=0
MOVL C00678 V=800.0 PL=0
MOVL C00679 V=800.0 PL=0
MOVL C00680 V=800.0 PL=0
MOVL C00681 V=800.0 PL=0
MOVL C00682 V=800.0 PL=0
MOVL C00683 V=800.0 PL=0
MOVL C00684 V=800.0 PL=0
MOVL C00685 V=800.0 PL=0
MOVL C00686 V=800.0 PL=0
MOVL C00687 V=800.0 PL=0
MOVL C00688 V=800.0 PL=0
MOVL C00689 V=800.0 PL=0
MOVL C00690 V=800.0 PL=0
MOVL C00691 V=800.0 PL=0
MOVL C00692 V=800.0 PL=0
MOVL C00693 V=800.0 PL=0
MOVL C00694 V=800.0 PL=0
MOVL C00695 V=800.0 PL=0
MOVL C00696 V=800.0 PL=0
MOVL C00697 V=800.0 PL=0
MOVL C00698 V=800.0 PL=0
MOVL C00699 V=800.0 PL=0
MOVL C00700 V=800.0 PL=0
MOVL C00701 V=800.0 PL=0
MOVL C00702 V=800.0 PL=0
MOVL C00703 V=800.0 PL=0
MOVL C00704 V=800.0 PL=0
MOVL C00705 V=800.0 PL=0
MOVL C00706 V=800.0 PL=0
MOVL C00707 V=800.0 PL=0
MOVL C00708 V=800.0 PL=0
MOVL C00709 V=800.0 PL=0
MOVL C00710 V=800.0 PL=0
MOVL C00711 V=800.0 PL=0
MOVL C00712 V=800.0 PL=0
MOVL C00713 V=800.0 PL=0
MOVL C00714 V=800.0 PL=0
MOVL C00715 V=800.0 PL=0
MOVL C00716 V=800.0 PL=0
MOVL C00717 V=800.0 PL=0
MOVL C00718 V=800.0 PL=0
MOVL C00719 V=800.0 PL=0
MOVL C00720 V=800.0 PL=0
MOVL C00721 V=800.0 PL=0
MOVL C00722 V=800.0 PL=0
MOVL C00723 V=800.0 PL=0
MOVL C00724 V=800.0 PL=0
MOVL C00725 V=800.0 PL=0
MOVL C00726 V=800.0 PL=0
MOVL C00727 V=800.0 PL=0
MOVL C00728 V=800.0 PL=0
MOVL C00729 V=800.0 PL=0
MOVL C00730 V=800.0 PL=0
MOVL C00731 V=800.0 PL=0
MOVL C00732 V=800.0 PL=0
MOVL C00733 V=800.0 PL=0
MOVL C00734 V=800.0 PL=0
MOVL C00735 V=800.0 PL=0
MOVL C00736 V=800.0 PL=0
MOVL C00737 V=800.0 PL=0
MOVL C00738 V=800.0 PL=0
MOVL C00739 V=800.0 PL=0
MOVL C00740 V=800.0 PL=0
MOVL C00741 V=800.0 PL=0
MOVL C00742 V=800.0 PL=0
MOVL C00743 V=800.0 PL=0
MOVL C00744 V=800.0 PL=0
MOVL C00745 V=800.0 PL=0
MOVL C00746 V=800.0 PL=0
MOVL C00747 V=800.0 PL=0
MOVL C00748 V=800.0 PL=0
MOVL C00749 V=800.0 PL=0
MOVL C00750 V=800.0 PL=0
MOVL C00751 V=800.0 PL=0
MOVL C00752 V=800.0 PL=0
MOVL C00753 V=800.0 PL=0
MOVL C00754 V=800.0 PL=0
MOVL C00755 V=800.0 PL=0
MOVL C00756 V=800.0 PL=0
MOVL C00757 V=800.0 PL=0
MOVL C00758 V=800.0 PL=0
MOVL C00759 V=800.0 PL=0
MOVL C00760 V=800.0 PL=0
MOVL C00761 V=800.0 PL=0
MOVL C00762 V=800.0 PL=0
MOVL C00763 V=800.0 PL=0
MOVL C00764 V=800.0 PL=0
MOVL C00765 V=800.0 PL=0
MOVL C00766 V=800.0 PL=0
MOVL C00767 V=800.0 PL=0
MOVL C00768 V=800.0 PL=0
MOVL C00769 V=800.0 PL=0
MOVL C00770 V=800.0 PL=0
MOVL C00771 V=800.0 PL=0
MOVL C00772 V=800.0 PL=0
MOVL C00773 V=800.0 PL=0
MOVL C00774 V=800.0 PL=0
MOVL C00775 V=800.0 PL=0
MOVL C00776 V=800.0 PL=0
MOVL C00777 V=800.0 PL=0
MOVL C00778 V=800.0 PL=0
MOVL C00779 V=800.0 PL=0
MOVL C00780 V=800.0 PL=0
MOVL C00781 V=800.0 PL=0
MOVL C00782 V=800.0 PL=0
MOVL C00783 V=800.0 PL=0
MOVL C00784 V=800.0 PL=0
MOVL C00785 V=800.0 PL=0
MOVL C00786 V=800.0 PL=0
MOVL C00787 V=800.0 PL=0
MOVL C00788 V=800.0 PL=0
MOVL C00789 V=800.0 PL=0
MOVL C00790 V=800.0 PL=0
MOVL C00791 V=800.0 PL=0
MOVL C00792 V=800.0 PL=0
MOVL C00793 V=800.0 PL=0
MOVL C00794 V=800.0 PL=0
MOVL C00795 V=800.0 PL=0
MOVL C00796 V=800.0 PL=0
MOVL C00797 V=800.0 PL=0
MOVL C00798 V=800.0 PL=0
MOVL C00799 V=800.0 PL=0
MOVL C00800 V=800.0 PL=0
MOVL C00801 V=800.0 PL=0
MOVL C00802 V=800.0 PL=0
MOVL C00803 V=800.0 PL=0
MOVL C00804 V=800.0 PL=0
MOVL C00805 V=800.0 PL=0
MOVL C00806 V=800.0 PL=0
MOVL C00807 V=800.0 PL=0
MOVL C00808 V=800.0 PL=0
MOVL C00809 V=800.0 PL=0
MOVL C00810 V=800.0 PL=0
MOVL C00811 V=800.0 PL=0
MOVL C00812 V=800.0 PL=0
MOVL C00813 V=800.0 PL=0
MOVL C00814 V=800.0 PL=0
MOVL C00815 V=800.0 PL=0
MOVL C00816 V=800.0 PL=0
MOVL C00817 V=800.0 PL=0
MOVL C00818 V=800.0 PL=0
MOVL C00819 V=800.0 PL=0
MOVL C00820 V=800.0 PL=0
MOVL C00821 V=800.0 PL=0
MOVL C00822 V=800.0 PL=0
MOVL C00823 V=800.0 PL=0
MOVL C00824 V=800.0 PL=0
MOVL C00825 V=800.0 PL=0
MOVL C00826 V=800.0 PL=0
MOVL C00827 V=800.0 PL=0
MOVL C00828 V=800.0 PL=0
MOVL C00829 V=800.0 PL=0
MOVL C00830 V=800.0 PL=0
MOVL C00831 V=800.0 PL=0
MOVL C00832 V=800.0 PL=0
MOVL C00833 V=800.0 PL=0
MOVL C00834 V=800.0 PL=0
MOVL C00835 V=800.0 PL=0
MOVL C00836 V=800.0 PL=0
MOVL C00837 V=800.0 PL=0
MOVL C00838 V=800.0 PL=0
MOVL C00839 V=800.0 PL=0
MOVL C00840 V=800.0 PL=0
MOVL C00841 V=800.0 PL=0
MOVL C00842 V=800.0 PL=0
MOVL C00843 V=800.0 PL=0
MOVL C00844 V=800.0 PL=0
MOVL C00845 V=800.0 PL=0
MOVL C00846 V=800.0 PL=0
MOVL C00847 V=800.0 PL=0
MOVL C00848 V=800.0 PL=0
MOVL C00849 V=800.0 PL=0
MOVL C00850 V=800.0 PL=0
MOVL C00851 V=800.0 PL=0
MOVL C00852 V=800.0 PL=0
MOVL C00853 V=800.0 PL=0
MOVL C00854 V=800.0 PL=0
MOVL C00855 V=800.0 PL=0
MOVL C00856 V=800.0 PL=0
MOVL C00857 V=800.0 PL=0
MOVL C00858 V=800.0 PL=0
MOVL C00859 V=800.0 PL=0
MOVL C00860 V=800.0 PL=0
MOVL C00861 V=800.0 PL=0
MOVL C00862 V=800.0 PL=0
MOVL C00863 V=800.0 PL=0
MOVL C00864 V=800.0 PL=0
MOVL C00865 V=800.0 PL=0
MOVL C00866 V=800.0 PL=0
MOVL C00867 V=800.0 PL=0
MOVL C00868 V=800.0 PL=0
MOVL C00869 V=800.0 PL=0
MOVL C00870 V=800.0 PL=0
MOVL C00871 V=800.0 PL=0
MOVL C00872 V=800.0 PL=0
MOVL C00873 V=800.0 PL=0
MOVL C00874 V=800.0 PL=0
MOVL C00875 V=800.0 PL=0
MOVL C00876 V=800.0 PL=0
MOVL C00877 V=800.0 PL=0
MOVL C00878 V=800.0 PL=0
MOVL C00879 V=800.0 PL=0
MOVL C00880 V=800.0 PL=0
MOVL C00881 V=800.0 PL=0
MOVL C00882 V=800.0 PL=0
MOVL C00883 V=800.0 PL=0
MOVL C00884 V=800.0 PL=0
MOVL C00885 V=800.0 PL=0
MOVL C00886 V=800.0 PL=0
MOVL C00887 V=800.0 PL=0
MOVL C00888 V=800.0 PL=0
MOVL C00889 V=800.0 PL=0
MOVL C00890 V=800.0 PL=0
MOVL C00891 V=800.0 PL=0
MOVL C00892 V=800.0 PL=0
MOVL C00893 V=800.0 PL=0
MOVL C00894 V=800.0 PL=0
MOVL C00895 V=800.0 PL=0
MOVL C00896 V=800.0 PL=0
MOVL C00897 V=800.0 PL=0
MOVL C00898 V=800.0 PL=0
MOVL C00899 V=800.0 PL=0
MOVL C00900 V=800.0 PL=0
MOVL C00901 V=800.0 PL=0
MOVL C00902 V=800.0 PL=0
MOVL C00903 V=800.0 PL=0
MOVL C00904 V=800.0 PL=0
MOVL C00905 V=800.0 PL=0
MOVL C00906 V=800.0 PL=0
MOVL C00907 V=800.0 PL=0
MOVL C00908 V=800.0 PL=0
MOVL C00909 V=800.0 PL=0
MOVL C00910 V=800.0 PL=0
MOVL C00911 V=800.0 PL=0
MOVL C00912 V=800.0 PL=0
MOVL C00913 V=800.0 PL=0
MOVL C00914 V=800.0 PL=0
MOVL C00915 V=800.0 PL=0
MOVL C00916 V=800.0 PL=0
MOVL C00917 V=800.0 PL=0
MOVL C00918 V=800.0 PL=0
MOVL C00919 V=800.0 PL=0
MOVL C00920 V=800.0 PL=0
MOVL C00921 V=800.0 PL=0
MOVL C00922 V=800.0 PL=0
MOVL C00923 V=800.0 PL=0
MOVL C00924 V=800.0 PL=0
MOVL C00925 V=800.0 PL=0
MOVL C00926 V=800.0 PL=0
MOVL C00927 V=800.0 PL=0
MOVL C00928 V=800.0 PL=0
MOVL C00929 V=800.0 PL=0
MOVL C00930 V=800.0 PL=0
MOVL C00931 V=800.0 PL=0
MOVL C00932 V=800.0 PL=0
MOVL C00933 V=800.0 PL=0
MOVL C00934 V=800.0 PL=0
MOVL C00935 V=800.0 PL=0
MOVL C00936 V=800.0 PL=0
MOVL C00937 V=800.0 PL=0
MOVL C00938 V=800.0 PL=0
MOVL C00939 V=800.0 PL=0
MOVL C00940 V=800.0 PL=0
MOVL C00941 V=800.0 PL=0
MOVL C00942 V=800.0 PL=0
MOVL C00943 V=800.0 PL=0
MOVL C00944 V=800.0 PL=0
MOVL C00945 V=800.0 PL=0
MOVL C00946 V=800.0 PL=0
MOVL C00947 V=800.0 PL=0
MOVL C00948 V=800.0 PL=0
MOVL C00949 V=800.0 PL=0
MOVL C00950 V=800.0 PL=0
MOVL C00951 V=800.0 PL=0
MOVL C00952 V=800.0 PL=0
MOVL C00953 V=800.0 PL=0
MOVL C00954 V=800.0 PL=0
MOVL C00955 V=800.0 PL=0
MOVL C00956 V=800.0 PL=0
MOVL C00957 V=800.0 PL=0
MOVL C00958 V=800.0 PL=0
MOVL C00959 V=800.0 PL=0
MOVL C00960 V=800.0 PL=0
MOVL C00961 V=800.0 PL=0
MOVL C00962 V=800.0 PL=0
MOVL C00963 V=800.0 PL=0
MOVL C00964 V=800.0 PL=0
MOVL C00965 V=800.0 PL=0
MOVL C00966 V=800.0 PL=0
MOVL C00967 V=800.0 PL=0
MOVL C00968 V=800.0 PL=0
MOVL C00969 V=800.0 PL=0
MOVL C00970 V=800.0 PL=0
MOVL C00971 V=800.0 PL=0
MOVL C00972 V=800.0 PL=0
MOVL C00973 V=800.0 PL=0
MOVL C00974 V=800.0 PL=0
MOVL C00975 V=800.0 PL=0
MOVL C00976 V=800.0 PL=0
MOVL C00977 V=800.0 PL=0
MOVL C00978 V=800.0 PL=0
MOVL C00979 V=800.0 PL=0
MOVL C00980 V=800.0 PL=0
MOVL C00981 V=800.0 PL=0
MOVL C00982 V=800.0 PL=0
MOVL C00983 V=800.0 PL=0
MOVL C00984 V=800.0 PL=0
MOVL C00985 V=800.0 PL=0
MOVL C00986 V=800.0 PL=0
MOVL C00987 V=800.0 PL=0
MOVL C00988 V=800.0 PL=0
MOVL C00989 V=800.0 PL=0
MOVL C00990 V=800.0 PL=0
MOVL C00991 V=800.0 PL=0
MOVL C00992 V=800.0 PL=0
MOVL C00993 V=800.0 PL=0
MOVL C00994 V=800.0 PL=0
MOVL C00995 V=800.0 PL=0
MOVL C00996 V=800.0 PL=0
MOVL C00997 V=800.0 PL=0
MOVL C00998 V=800.0 PL=0
MOVL C00999 V=800.0 PL=0
MOVL C01000 V=800.0 PL=0
MOVL C01001 V=800.0 PL=0
MOVL C01002 V=800.0 PL=0
MOVL C01003 V=800.0 PL=0
MOVL C01004 V=800.0 PL=0
MOVL C01005 V=800.0 PL=0
MOVL C01006 V=800.0 PL=0
MOVL C01007 V=800.0 PL=0
MOVL C01008 V=800.0 PL=0
MOVL C01009 V=800.0 PL=0
MOVL C01010 V=800.0 PL=0
MOVL C01011 V=800.0 PL=0
MOVL C01012 V=800.0 PL=0
MOVL C01013 V=800.0 PL=0
MOVL C01014 V=800.0 PL=0
MOVL C01015 V=800.0 PL=0
MOVL C01016 V=800.0 PL=0
MOVL C01017 V=800.0 PL=0
MOVL C01018 V=800.0 PL=0
MOVL C01019 V=800.0 PL=0
MOVL C01020 V=800.0 PL=0
MOVL C01021 V=800.0 PL=0
MOVL C01022 V=800.0 PL=0
MOVL C01023 V=800.0 PL=0
MOVL C01024 V=800.0 PL=0
MOVL C01025 V=800.0 PL=0
MOVL C01026 V=800.0 PL=0
MOVL C01027 V=800.0 PL=0
MOVL C01028 V=800.0 PL=0
MOVL C01029 V=800.0 PL=0
MOVL C01030 V=800.0 PL=0
MOVL C01031 V=800.0 PL=0
MOVL C01032 V=800.0 PL=0
MOVL C01033 V=800.0 PL=0
MOVL C01034 V=800.0 PL=0
MOVL C01035 V=800.0 PL=0
MOVL C01036 V=800.0 PL=0
MOVL C01037 V=800.0 PL=0
MOVL C01038 V=800.0 PL=0
MOVL C01039 V=800.0 PL=0
MOVL C01040 V=800.0 PL=0
MOVL C01041 V=800.0 PL=0
MOVL C01042 V=800.0 PL=0
MOVL C01043 V=800.0 PL=0
MOVL C01044 V=800.0 PL=0
MOVL C01045 V=800.0 PL=0
MOVL C01046 V=800.0 PL=0
MOVL C01047 V=800.0 PL=0
MOVL C01048 V=800.0 PL=0
MOVL C01049 V=800.0 PL=0
MOVL C01050 V=800.0 PL=0
MOVL C01051 V=800.0 PL=0
MOVL C01052 V=800.0 PL=0
MOVL C01053 V=800.0 PL=0
MOVL C01054 V=800.0 PL=0
MOVL C01055 V=800.0 PL=0
MOVL C01056 V=800.0 PL=0
MOVL C01057 V=800.0 PL=0
MOVL C01058 V=800.0 PL=0
MOVL C01059 V=800.0 PL=0
MOVL C01060 V=800.0 PL=0
MOVL C01061 V=800.0 PL=0
MOVL C01062 V=800.0 PL=0
MOVL C01063 V=800.0 PL=0
MOVL C01064 V=800.0 PL=0
MOVL C01065 V=800.0 PL=0
MOVL C01066 V=800.0 PL=0
MOVL C01067 V=800.0 PL=0
MOVL C01068 V=800.0 PL=0
MOVL C01069 V=800.0 PL=0
MOVL C01070 V=800.0 PL=0
MOVL C01071 V=800.0 PL=0
MOVL C01072 V=800.0 PL=0
MOVL C01073 V=800.0 PL=0
MOVL C01074 V=800.0 PL=0
MOVL C01075 V=800.0 PL=0
MOVL C01076 V=800.0 PL=0
MOVL C01077 V=800.0 PL=0
MOVL C01078 V=800.0 PL=0
MOVL C01079 V=800.0 PL=0
MOVL C01080 V=800.0 PL=0
MOVL C01081 V=800.0 PL=0
MOVL C01082 V=800.0 PL=0
MOVL C01083 V=800.0 PL=0
MOVL C01084 V=800.0 PL=0
MOVL C01085 V=800.0 PL=0
MOVL C01086 V=800.0 PL=0
MOVL C01087 V=800.0 PL=0
MOVL C01088 V=800.0 PL=0
MOVL C01089 V=800.0 PL=0
MOVL C01090 V=800.0 PL=0
MOVL C01091 V=800.0 PL=0
MOVL C01092 V=800.0 PL=0
MOVL C01093 V=800.0 PL=0
MOVL C01094 V=800.0 PL=0
MOVL C01095 V=800.0 PL=0
MOVL C01096 V=800.0 PL=0
MOVL C01097 V=800.0 PL=0
MOVL C01098 V=800.0 PL=0
MOVL C01099 V=800.0 PL=0
MOVL C01100 V=800.0 PL=0
MOVL C01101 V=800.0 PL=0
MOVL C01102 V=800.0 PL=0
MOVL C01103 V=800.0 PL=0
MOVL C01104 V=800.0 PL=0
MOVL C01105 V=800.0 PL=0
MOVL C01106 V=800.0 PL=0
MOVL C01107 V=800.0 PL=0
MOVL C01108 V=800.0 PL=0
MOVL C01109 V=800.0 PL=0
MOVL C01110 V=800.0 PL=0
MOVL C01111 V=800.0 PL=0
MOVL C01112 V=800.0 PL=0
MOVL C01113 V=800.0 PL=0
MOVL C01114 V=800.0 PL=0
MOVL C01115 V=800.0 PL=0
MOVL C01116 V=800.0 PL=0
MOVL C01117 V=800.0 PL=0
MOVL C01118 V=800.0 PL=0
MOVL C01119 V=800.0 PL=0
MOVL C01120 V=800.0 PL=0
MOVL C01121 V=800.0 PL=0
MOVL C01122 V=800.0 PL=0
MOVL C01123 V=800.0 PL=0
MOVL C01124 V=800.0 PL=0
MOVL C01125 V=800.0 PL=0
MOVL C01126 V=800.0 PL=0
MOVL C01127 V=800.0 PL=0
MOVL C01128 V=800.0 PL=0
MOVL C01129 V=800.0 PL=0
MOVL C01130 V=800.0 PL=0
MOVL C01131 V=800.0 PL=0
MOVL C01132 V=800.0 PL=0
MOVL C01133 V=800.0 PL=0
MOVL C01134 V=800.0 PL=0
MOVL C01135 V=800.0 PL=0
MOVL C01136 V=800.0 PL=0
MOVL C01137 V=800.0 PL=0
MOVL C01138 V=800.0 PL=0
MOVL C01139 V=800.0 PL=0
MOVL C01140 V=800.0 PL=0
MOVL C01141 V=800.0 PL=0
MOVL C01142 V=800.0 PL=0
MOVL C01143 V=800.0 PL=0
MOVL C01144 V=800.0 PL=0
MOVL C01145 V=800.0 PL=0
MOVL C01146 V=800.0 PL=0
MOVL C01147 V=800.0 PL=0
MOVL C01148 V=800.0 PL=0
MOVL C01149 V=800.0 PL=0
MOVL C01150 V=800.0 PL=0
MOVL C01151 V=800.0 PL=0
MOVL C01152 V=800.0 PL=0
MOVL C01153 V=800.0 PL=0
MOVL C01154 V=800.0 PL=0
MOVL C01155 V=800.0 PL=0
MOVL C01156 V=800.0 PL=0
MOVL C01157 V=800.0 PL=0
MOVL C01158 V=800.0 PL=0
MOVL C01159 V=800.0 PL=0
MOVL C01160 V=800.0 PL=0
MOVL C01161 V=800.0 PL=0
MOVL C01162 V=800.0 PL=0
MOVL C01163 V=800.0 PL=0
MOVL C01164 V=800.0 PL=0
MOVL C01165 V=800.0 PL=0
MOVL C01166 V=800.0 PL=0
MOVL C01167 V=800.0 PL=0
MOVL C01168 V=800.0 PL=0
MOVL C01169 V=800.0 PL=0
MOVL C01170 V=800.0 PL=0
MOVL C01171 V=800.0 PL=0
MOVL C01172 V=800.0 PL=0
MOVL C01173 V=800.0 PL=0
MOVL C01174 V=800.0 PL=0
MOVL C01175 V=800.0 PL=0
MOVL C01176 V=800.0 PL=0
MOVL C01177 V=800.0 PL=0
MOVL C01178 V=800.0 PL=0
MOVL C01179 V=800.0 PL=0
MOVL C01180 V=800.0 PL=0
MOVL C01181 V=800.0 PL=0
MOVL C01182 V=800.0 PL=0
MOVL C01183 V=800.0 PL=0
MOVL C01184 V=800.0 PL=0
MOVL C01185 V=800.0 PL=0
MOVL C01186 V=800.0 PL=0
MOVL C01187 V=800.0 PL=0
MOVL C01188 V=800.0 PL=0
MOVL C01189 V=800.0 PL=0
MOVL C01190 V=800.0 PL=0
MOVL C01191 V=800.0 PL=0
MOVL C01192 V=800.0 PL=0
MOVL C01193 V=800.0 PL=0
MOVL C01194 V=800.0 PL=0
MOVL C01195 V=800.0 PL=0
MOVL C01196 V=800.0 PL=0
MOVL C01197 V=800.0 PL=0
MOVL C01198 V=800.0 PL=0
MOVL C01199 V=800.0 PL=0
MOVL C01200 V=800.0 PL=0
MOVL C01201 V=800.0 PL=0
MOVL C01202 V=800.0 PL=0
MOVL C01203 V=800.0 PL=0
MOVL C01204 V=800.0 PL=0
MOVL C01205 V=800.0 PL=0
MOVL C01206 V=800.0 PL=0
MOVL C01207 V=800.0 PL=0
MOVL C01208 V=800.0 PL=0
MOVL C01209 V=800.0 PL=0
MOVL C01210 V=800.0 PL=0
MOVL C01211 V=800.0 PL=0
MOVL C01212 V=800.0 PL=0
MOVL C01213 V=800.0 PL=0
MOVL C01214 V=800.0 PL=0
MOVL C01215 V=800.0 PL=0
MOVL C01216 V=800.0 PL=0
MOVL C01217 V=800.0 PL=0
MOVL C01218 V=800.0 PL=0
MOVL C01219 V=800.0 PL=0
MOVL C01220 V=800.0 PL=0
MOVL C01221 V=800.0 PL=0
MOVL C01222 V=800.0 PL=0
MOVL C01223 V=800.0 PL=0
MOVL C01224 V=800.0 PL=0
MOVL C01225 V=800.0 PL=0
MOVL C01226 V=800.0 PL=0
MOVL C01227 V=800.0 PL=0
MOVL C01228 V=800.0 PL=0
MOVL C01229 V=800.0 PL=0
MOVL C01230 V=800.0 PL=0
MOVL C01231 V=800.0 PL=0
MOVL C01232 V=800.0 PL=0
MOVL C01233 V=800.0 PL=0
MOVL C01234 V=800.0 PL=0
MOVL C01235 V=800.0 PL=0
MOVL C01236 V=800.0 PL=0
MOVL C01237 V=800.0 PL=0
MOVL C01238 V=800.0 PL=0
MOVL C01239 V=800.0 PL=0
MOVL C01240 V=800.0 PL=0
MOVL C01241 V=800.0 PL=0
MOVL C01242 V=800.0 PL=0
MOVL C01243 V=800.0 PL=0
MOVL C01244 V=800.0 PL=0
MOVL C01245 V=800.0 PL=0
MOVL C01246 V=800.0 PL=0
MOVL C01247 V=800.0 PL=0
MOVL C01248 V=800.0 PL=0
MOVL C01249 V=800.0 PL=0
MOVL C01250 V=800.0 PL=0
MOVL C01251 V=800.0 PL=0
MOVL C01252 V=800.0 PL=0
MOVL C01253 V=800.0 PL=0
MOVL C01254 V=800.0 PL=0
MOVL C01255 V=800.0 PL=0
MOVL C01256 V=800.0 PL=0
MOVL C01257 V=800.0 PL=0
MOVL C01258 V=800.0 PL=0
MOVL C01259 V=800.0 PL=0
MOVL C01260 V=800.0 PL=0
MOVL C01261 V=800.0 PL=0
MOVL C01262 V=800.0 PL=0
MOVL C01263 V=800.0 PL=0
MOVL C01264 V=800.0 PL=0
MOVL C01265 V=800.0 PL=0
MOVL C01266 V=800.0 PL=0
MOVL C01267 V=800.0 PL=0
MOVL C01268 V=800.0 PL=0
MOVL C01269 V=800.0 PL=0
MOVL C01270 V=800.0 PL=0
MOVL C01271 V=800.0 PL=0
MOVL C01272 V=800.0 PL=0
MOVL C01273 V=800.0 PL=0
MOVL C01274 V=800.0 PL=0
MOVL C01275 V=800.0 PL=0
MOVL C01276 V=800.0 PL=0
MOVL C01277 V=800.0 PL=0
MOVL C01278 V=800.0 PL=0
MOVL C01279 V=800.0 PL=0
MOVL C01280 V=800.0 PL=0
MOVL C01281 V=800.0 PL=0
MOVL C01282 V=800.0 PL=0
MOVL C01283 V=800.0 PL=0
MOVL C01284 V=800.0 PL=0
MOVL C01285 V=800.0 PL=0
MOVL C01286 V=800.0 PL=0
MOVL C01287 V=800.0 PL=0
MOVL C01288 V=800.0 PL=0
MOVL C01289 V=800.0 PL=0
MOVL C01290 V=800.0 PL=0
MOVL C01291 V=800.0 PL=0
MOVL C01292 V=800.0 PL=0
MOVL C01293 V=800.0 PL=0
MOVL C01294 V=800.0 PL=0
MOVL C01295 V=800.0 PL=0
MOVL C01296 V=800.0 PL=0
MOVL C01297 V=800.0 PL=0
MOVL C01298 V=800.0 PL=0
MOVL C01299 V=800.0 PL=0
MOVL C01300 V=800.0 PL=0
MOVL C01301 V=800.0 PL=0
MOVL C01302 V=800.0 PL=0
MOVL C01303 V=800.0 PL=0
MOVL C01304 V=800.0 PL=0
MOVL C01305 V=800.0 PL=0
MOVL C01306 V=800.0 PL=0
MOVL C01307 V=800.0 PL=0
MOVL C01308 V=800.0 PL=0
MOVL C01309 V=800.0 PL=0
MOVL C01310 V=800.0 PL=0
MOVL C01311 V=800.0 PL=0
MOVL C01312 V=800.0 PL=0
MOVL C01313 V=800.0 PL=0
MOVL C01314 V=800.0 PL=0
MOVL C01315 V=800.0 PL=0
MOVL C01316 V=800.0 PL=0
MOVL C01317 V=800.0 PL=0
MOVL C01318 V=800.0 PL=0
MOVL C01319 V=800.0 PL=0
MOVL C01320 V=800.0 PL=0
MOVL C01321 V=800.0 PL=0
MOVL C01322 V=800.0 PL=0
MOVL C01323 V=800.0 PL=0
MOVL C01324 V=800.0 PL=0
MOVL C01325 V=800.0 PL=0
MOVL C01326 V=800.0 PL=0
MOVL C01327 V=800.0 PL=0
MOVL C01328 V=800.0 PL=0
MOVL C01329 V=800.0 PL=0
MOVL C01330 V=800.0 PL=0
MOVL C01331 V=800.0 PL=0
MOVL C01332 V=800.0 PL=0
MOVL C01333 V=800.0 PL=0
MOVL C01334 V=800.0 PL=0
MOVL C01335 V=800.0 PL=0
MOVL C01336 V=800.0 PL=0
MOVL C01337 V=800.0 PL=0
MOVL C01338 V=800.0 PL=0
MOVL C01339 V=800.0 PL=0
MOVL C01340 V=800.0 PL=0
MOVL C01341 V=800.0 PL=0
MOVL C01342 V=800.0 PL=0
MOVL C01343 V=800.0 PL=0
MOVL C01344 V=800.0 PL=0
MOVL C01345 V=800.0 PL=0
MOVL C01346 V=800.0 PL=0
MOVL C01347 V=800.0 PL=0
MOVL C01348 V=800.0 PL=0
MOVL C01349 V=800.0 PL=0
MOVL C01350 V=800.0 PL=0
MOVL C01351 V=800.0 PL=0
MOVL C01352 V=800.0 PL=0
MOVL C01353 V=800.0 PL=0
MOVL C01354 V=800.0 PL=0
MOVL C01355 V=800.0 PL=0
MOVL C01356 V=800.0 PL=0
MOVL C01357 V=800.0 PL=0
MOVL C01358 V=800.0 PL=0
MOVL C01359 V=800.0 PL=0
MOVL C01360 V=800.0 PL=0
MOVL C01361 V=800.0 PL=0
MOVL C01362 V=800.0 PL=0
MOVL C01363 V=800.0 PL=0
MOVL C01364 V=800.0 PL=0
MOVL C01365 V=800.0 PL=0
MOVL C01366 V=800.0 PL=0
MOVL C01367 V=800.0 PL=0
MOVL C01368 V=800.0 PL=0
MOVL C01369 V=800.0 PL=0
MOVL C01370 V=800.0 PL=0
MOVL C01371 V=800.0 PL=0
MOVL C01372 V=800.0 PL=0
MOVL C01373 V=800.0 PL=0
MOVL C01374 V=800.0 PL=0
MOVL C01375 V=800.0 PL=0
MOVL C01376 V=800.0 PL=0
MOVL C01377 V=800.0 PL=0
MOVL C01378 V=800.0 PL=0
MOVL C01379 V=800.0 PL=0
MOVL C01380 V=800.0 PL=0
MOVL C01381 V=800.0 PL=0
MOVL C01382 V=800.0 PL=0
MOVL C01383 V=800.0 PL=0
MOVL C01384 V=800.0 PL=0
MOVL C01385 V=800.0 PL=0
MOVL C01386 V=800.0 PL=0
MOVL C01387 V=800.0 PL=0
MOVL C01388 V=800.0 PL=0
MOVL C01389 V=800.0 PL=0
MOVL C01390 V=800.0 PL=0
MOVL C01391 V=800.0 PL=0
MOVL C01392 V=800.0 PL=0
MOVL C01393 V=800.0 PL=0
MOVL C01394 V=800.0 PL=0
MOVL C01395 V=800.0 PL=0
MOVL C01396 V=800.0 PL=0
MOVL C01397 V=800.0 PL=0
MOVL C01398 V=800.0 PL=0
MOVL C01399 V=800.0 PL=0
MOVL C01400 V=800.0 PL=0
MOVL C01401 V=800.0 PL=0
MOVL C01402 V=800.0 PL=0
MOVL C01403 V=800.0 PL=0
MOVL C01404 V=800.0 PL=0
MOVL C01405 V=800.0 PL=0
MOVL C01406 V=800.0 PL=0
MOVL C01407 V=800.0 PL=0
MOVL C01408 V=800.0 PL=0
MOVL C01409 V=800.0 PL=0
MOVL C01410 V=800.0 PL=0
MOVL C01411 V=800.0 PL=0
MOVL C01412 V=800.0 PL=0
MOVL C01413 V=800.0 PL=0
MOVL C01414 V=800.0 PL=0
MOVL C01415 V=800.0 PL=0
MOVL C01416 V=800.0 PL=0
MOVL C01417 V=800.0 PL=0
MOVL C01418 V=800.0 PL=0
MOVL C01419 V=800.0 PL=0
MOVL C01420 V=800.0 PL=0
MOVL C01421 V=800.0 PL=0
MOVL C01422 V=800.0 PL=0
MOVL C01423 V=800.0 PL=0
MOVL C01424 V=800.0 PL=0
MOVL C01425 V=800.0 PL=0
MOVL C01426 V=800.0 PL=0
MOVL C01427 V=800.0 PL=0
MOVL C01428 V=800.0 PL=0
MOVL C01429 V=800.0 PL=0
MOVL C01430 V=800.0 PL=0
MOVL C01431 V=800.0 PL=0
MOVL C01432 V=800.0 PL=0
MOVL C01433 V=800.0 PL=0
MOVL C01434 V=800.0 PL=0
MOVL C01435 V=800.0 PL=0
MOVL C01436 V=800.0 PL=0
MOVL C01437 V=800.0 PL=0
MOVL C01438 V=800.0 PL=0
MOVL C01439 V=800.0 PL=0
MOVL C01440 V=800.0 PL=0
MOVL C01441 V=800.0 PL=0
MOVL C01442 V=800.0 PL=0
MOVL C01443 V=800.0 PL=0
MOVL C01444 V=800.0 PL=0
MOVL C01445 V=800.0 PL=0
MOVL C01446 V=800.0 PL=0
MOVL C01447 V=800.0 PL=0
MOVL C01448 V=800.0 PL=0
MOVL C01449 V=800.0 PL=0
MOVL C01450 V=800.0 PL=0
MOVL C01451 V=800.0 PL=0
MOVL C01452 V=800.0 PL=0
MOVL C01453 V=800.0 PL=0
MOVL C01454 V=800.0 PL=0
MOVL C01455 V=800.0 PL=0
MOVL C01456 V=800.0 PL=0
MOVL C01457 V=800.0 PL=0
MOVL C01458 V=800.0 PL=0
MOVL C01459 V=800.0 PL=0
MOVL C01460 V=800.0 PL=0
MOVL C01461 V=800.0 PL=0
MOVL C01462 V=800.0 PL=0
MOVL C01463 V=800.0 PL=0
MOVL C01464 V=800.0 PL=0
MOVL C01465 V=800.0 PL=0
MOVL C01466 V=800.0 PL=0
MOVL C01467 V=800.0 PL=0
MOVL C01468 V=800.0 PL=0
MOVL C01469 V=800.0 PL=0
MOVL C01470 V=800.0 PL=0
MOVL C01471 V=800.0 PL=0
MOVL C01472 V=800.0 PL=0
MOVL C01473 V=800.0 PL=0
MOVL C01474 V=800.0 PL=0
MOVL C01475 V=800.0 PL=0
MOVL C01476 V=800.0 PL=0
MOVL C01477 V=800.0 PL=0
MOVL C01478 V=800.0 PL=0
MOVL C01479 V=800.0 PL=0
MOVL C01480 V=800.0 PL=0
MOVL C01481 V=800.0 PL=0
MOVL C01482 V=800.0 PL=0
MOVL C01483 V=800.0 PL=0
MOVL C01484 V=800.0 PL=0
MOVL C01485 V=800.0 PL=0
MOVL C01486 V=800.0 PL=0
MOVL C01487 V=800.0 PL=0
MOVL C01488 V=800.0 PL=0
MOVL C01489 V=800.0 PL=0
MOVL C01490 V=800.0 PL=0
MOVL C01491 V=800.0 PL=0
MOVL C01492 V=800.0 PL=0
MOVL C01493 V=800.0 PL=0
MOVL C01494 V=800.0 PL=0
MOVL C01495 V=800.0 PL=0
MOVL C01496 V=800.0 PL=0
MOVL C01497 V=800.0 PL=0
MOVL C01498 V=800.0 PL=0
MOVL C01499 V=800.0 PL=0
MOVL C01500 V=800.0 PL=0
MOVL C01501 V=800.0 PL=0
MOVL C01502 V=800.0 PL=0
MOVL C01503 V=800.0 PL=0
MOVL C01504 V=800.0 PL=0
MOVL C01505 V=800.0 PL=0
MOVL C01506 V=800.0 PL=0
MOVL C01507 V=800.0 PL=0
MOVL C01508 V=800.0 PL=0
MOVL C01509 V=800.0 PL=0
MOVL C01510 V=800.0 PL=0
MOVL C01511 V=800.0 PL=0
MOVL C01512 V=800.0 PL=0
MOVL C01513 V=800.0 PL=0
MOVL C01514 V=800.0 PL=0
MOVL C01515 V=800.0 PL=0
MOVL C01516 V=800.0 PL=0
MOVL C01517 V=800.0 PL=0
MOVL C01518 V=800.0 PL=0
MOVL C01519 V=800.0 PL=0
MOVL C01520 V=800.0 PL=0
MOVL C01521 V=800.0 PL=0
MOVL C01522 V=800.0 PL=0
MOVL C01523 V=800.0 PL=0
MOVL C01524 V=800.0 PL=0
MOVL C01525 V=800.0 PL=0
MOVL C01526 V=800.0 PL=0
MOVL C01527 V=800.0 PL=0
MOVL C01528 V=800.0 PL=0
MOVL C01529 V=800.0 PL=0
MOVL C01530 V=800.0 PL=0
MOVL C01531 V=800.0 PL=0
MOVL C01532 V=800.0 PL=0
MOVL C01533 V=800.0 PL=0
MOVL C01534 V=800.0 PL=0
MOVL C01535 V=800.0 PL=0
MOVL C01536 V=800.0 PL=0
MOVL C01537 V=800.0 PL=0
MOVL C01538 V=800.0 PL=0
MOVL C01539 V=800.0 PL=0
MOVL C01540 V=800.0 PL=0
MOVL C01541 V=800.0 PL=0
MOVL C01542 V=800.0 PL=0
MOVL C01543 V=800.0 PL=0
MOVL C01544 V=800.0 PL=0
MOVL C01545 V=800.0 PL=0
MOVL C01546 V=800.0 PL=0
MOVL C01547 V=800.0 PL=0
MOVL C01548 V=800.0 PL=0
MOVL C01549 V=800.0 PL=0
MOVL C01550 V=800.0 PL=0
MOVL C01551 V=800.0 PL=0
MOVL C01552 V=800.0 PL=0
MOVL C01553 V=800.0 PL=0
MOVL C01554 V=800.0 PL=0
MOVL C01555 V=800.0 PL=0
MOVL C01556 V=800.0 PL=0
MOVL C01557 V=800.0 PL=0
MOVL C01558 V=800.0 PL=0
MOVL C01559 V=800.0 PL=0
MOVL C01560 V=800.0 PL=0
MOVL C01561 V=800.0 PL=0
MOVL C01562 V=800.0 PL=0
MOVL C01563 V=800.0 PL=0
MOVL C01564 V=800.0 PL=0
MOVL C01565 V=800.0 PL=0
MOVL C01566 V=800.0 PL=0
MOVL C01567 V=800.0 PL=0
MOVL C01568 V=800.0 PL=0
MOVL C01569 V=800.0 PL=0
MOVL C01570 V=800.0 PL=0
MOVL C01571 V=800.0 PL=0
MOVL C01572 V=800.0 PL=0
MOVL C01573 V=800.0 PL=0
MOVL C01574 V=800.0 PL=0
MOVL C01575 V=800.0 PL=0
MOVL C01576 V=800.0 PL=0
MOVL C01577 V=800.0 PL=0
MOVL C01578 V=800.0 PL=0
MOVL C01579 V=800.0 PL=0
MOVL C01580 V=800.0 PL=0
MOVL C01581 V=800.0 PL=0
MOVL C01582 V=800.0 PL=0
MOVL C01583 V=800.0 PL=0
MOVL C01584 V=800.0 PL=0
MOVL C01585 V=800.0 PL=0
MOVL C01586 V=800.0 PL=0
MOVL C01587 V=800.0 PL=0
MOVL C01588 V=800.0 PL=0
MOVL C01589 V=800.0 PL=0
MOVL C01590 V=800.0 PL=0
MOVL C01591 V=800.0 PL=0
MOVL C01592 V=800.0 PL=0
MOVL C01593 V=800.0 PL=0
MOVL C01594 V=800.0 PL=0
MOVL C01595 V=800.0 PL=0
MOVL C01596 V=800.0 PL=0
MOVL C01597 V=800.0 PL=0
MOVL C01598 V=800.0 PL=0
MOVL C01599 V=800.0 PL=0
MOVL C01600 V=800.0 PL=0
MOVL C01601 V=800.0 PL=0
MOVL C01602 V=800.0 PL=0
MOVL C01603 V=800.0 PL=0
MOVL C01604 V=800.0 PL=0
MOVL C01605 V=800.0 PL=0
MOVL C01606 V=800.0 PL=0
MOVL C01607 V=800.0 PL=0
MOVL C01608 V=800.0 PL=0
MOVL C01609 V=800.0 PL=0
MOVL C01610 V=800.0 PL=0
MOVL C01611 V=800.0 PL=0
MOVL C01612 V=800.0 PL=0
MOVL C01613 V=800.0 PL=0
MOVL C01614 V=800.0 PL=0
MOVL C01615 V=800.0 PL=0
MOVL C01616 V=800.0 PL=0
MOVL C01617 V=800.0 PL=0
MOVL C01618 V=800.0 PL=0
MOVL C01619 V=800.0 PL=0
MOVL C01620 V=800.0 PL=0
MOVL C01621 V=800.0 PL=0
MOVL C01622 V=800.0 PL=0
MOVL C01623 V=800.0 PL=0
MOVL C01624 V=800.0 PL=0
MOVL C01625 V=800.0 PL=0
MOVL C01626 V=800.0 PL=0
MOVL C01627 V=800.0 PL=0
MOVL C01628 V=800.0 PL=0
MOVL C01629 V=800.0 PL=0
MOVL C01630 V=800.0 PL=0
MOVL C01631 V=800.0 PL=0
MOVL C01632 V=800.0 PL=0
MOVL C01633 V=800.0 PL=0
MOVL C01634 V=800.0 PL=0
MOVL C01635 V=800.0 PL=0
MOVL C01636 V=800.0 PL=0
MOVL C01637 V=800.0 PL=0
MOVL C01638 V=800.0 PL=0
MOVL C01639 V=800.0 PL=0
MOVL C01640 V=800.0 PL=0
MOVL C01641 V=800.0 PL=0
MOVL C01642 V=800.0 PL=0
MOVL C01643 V=800.0 PL=0
MOVL C01644 V=800.0 PL=0
MOVL C01645 V=800.0 PL=0
MOVL C01646 V=800.0 PL=0
MOVL C01647 V=800.0 PL=0
MOVL C01648 V=800.0 PL=0
MOVL C01649 V=800.0 PL=0
MOVL C01650 V=800.0 PL=0
MOVL C01651 V=800.0 PL=0
MOVL C01652 V=800.0 PL=0
MOVL C01653 V=800.0 PL=0
MOVL C01654 V=800.0 PL=0
MOVL C01655 V=800.0 PL=0
MOVL C01656 V=800.0 PL=0
MOVL C01657 V=800.0 PL=0
MOVL C01658 V=800.0 PL=0
MOVL C01659 V=800.0 PL=0
MOVL C01660 V=800.0 PL=0
MOVL C01661 V=800.0 PL=0
MOVL C01662 V=800.0 PL=0
MOVL C01663 V=800.0 PL=0
MOVL C01664 V=800.0 PL=0
MOVL C01665 V=800.0 PL=0
MOVL C01666 V=800.0 PL=0
MOVL C01667 V=800.0 PL=0
MOVL C01668 V=800.0 PL=0
MOVL C01669 V=800.0 PL=0
MOVL C01670 V=800.0 PL=0
MOVL C01671 V=800.0 PL=0
MOVL C01672 V=800.0 PL=0
MOVL C01673 V=800.0 PL=0
MOVL C01674 V=800.0 PL=0
MOVL C01675 V=800.0 PL=0
MOVL C01676 V=800.0 PL=0
MOVL C01677 V=800.0 PL=0
MOVL C01678 V=800.0 PL=0
MOVL C01679 V=800.0 PL=0
MOVL C01680 V=800.0 PL=0
MOVL C01681 V=800.0 PL=0
MOVL C01682 V=800.0 PL=0
MOVL C01683 V=800.0 PL=0
MOVL C01684 V=800.0 PL=0
MOVL C01685 V=800.0 PL=0
MOVL C01686 V=800.0 PL=0
MOVL C01687 V=800.0 PL=0
MOVL C01688 V=800.0 PL=0
MOVL C01689 V=800.0 PL=0
MOVL C01690 V=800.0 PL=0
MOVL C01691 V=800.0 PL=0
MOVL C01692 V=800.0 PL=0
MOVL C01693 V=800.0 PL=0
MOVL C01694 V=800.0 PL=0
MOVL C01695 V=800.0 PL=0
MOVL C01696 V=800.0 PL=0
MOVL C01697 V=800.0 PL=0
MOVL C01698 V=800.0 PL=0
MOVL C01699 V=800.0 PL=0
MOVL C01700 V=800.0 PL=0
MOVL C01701 V=800.0 PL=0
MOVL C01702 V=800.0 PL=0
MOVL C01703 V=800.0 PL=0
MOVL C01704 V=800.0 PL=0
MOVL C01705 V=800.0 PL=0
MOVL C01706 V=800.0 PL=0
MOVL C01707 V=800.0 PL=0
MOVL C01708 V=800.0 PL=0
MOVL C01709 V=800.0 PL=0
MOVL C01710 V=800.0 PL=0
MOVL C01711 V=800.0 PL=0
MOVL C01712 V=800.0 PL=0
MOVL C01713 V=800.0 PL=0
MOVL C01714 V=800.0 PL=0
MOVL C01715 V=800.0 PL=0
MOVL C01716 V=800.0 PL=0
MOVL C01717 V=800.0 PL=0
MOVL C01718 V=800.0 PL=0
MOVL C01719 V=800.0 PL=0
MOVL C01720 V=800.0 PL=0
MOVL C01721 V=800.0 PL=0
MOVL C01722 V=800.0 PL=0
MOVL C01723 V=800.0 PL=0
MOVL C01724 V=800.0 PL=0
MOVL C01725 V=800.0 PL=0
MOVL C01726 V=800.0 PL=0
MOVL C01727 V=800.0 PL=0
MOVL C01728 V=800.0 PL=0
MOVL C01729 V=800.0 PL=0
MOVL C01730 V=800.0 PL=0
MOVL C01731 V=800.0 PL=0
MOVL C01732 V=800.0 PL=0
MOVL C01733 V=800.0 PL=0
MOVL C01734 V=800.0 PL=0
MOVL C01735 V=800.0 PL=0
MOVL C01736 V=800.0 PL=0
MOVL C01737 V=800.0 PL=0
MOVL C01738 V=800.0 PL=0
MOVL C01739 V=800.0 PL=0
MOVL C01740 V=800.0 PL=0
MOVL C01741 V=800.0 PL=0
MOVL C01742 V=800.0 PL=0
MOVL C01743 V=800.0 PL=0
MOVL C01744 V=800.0 PL=0
MOVL C01745 V=800.0 PL=0
MOVL C01746 V=800.0 PL=0
MOVL C01747 V=800.0 PL=0
MOVL C01748 V=800.0 PL=0
MOVL C01749 V=800.0 PL=0
MOVL C01750 V=800.0 PL=0
MOVL C01751 V=800.0 PL=0
MOVL C01752 V=800.0 PL=0
MOVL C01753 V=800.0 PL=0
MOVL C01754 V=800.0 PL=0
MOVL C01755 V=800.0 PL=0
MOVL C01756 V=800.0 PL=0
MOVL C01757 V=800.0 PL=0
MOVL C01758 V=800.0 PL=0
MOVL C01759 V=800.0 PL=0
MOVL C01760 V=800.0 PL=0
MOVL C01761 V=800.0 PL=0
MOVL C01762 V=800.0 PL=0
MOVL C01763 V=800.0 PL=0
MOVL C01764 V=800.0 PL=0
MOVL C01765 V=800.0 PL=0
MOVL C01766 V=800.0 PL=0
MOVL C01767 V=800.0 PL=0
MOVL C01768 V=800.0 PL=0
MOVL C01769 V=800.0 PL=0
MOVL C01770 V=800.0 PL=0
MOVL C01771 V=800.0 PL=0
MOVL C01772 V=800.0 PL=0
MOVL C01773 V=800.0 PL=0
MOVL C01774 V=800.0 PL=0
MOVL C01775 V=800.0 PL=0
MOVL C01776 V=800.0 PL=0
MOVL C01777 V=800.0 PL=0
MOVL C01778 V=800.0 PL=0
MOVL C01779 V=800.0 PL=0
MOVL C01780 V=800.0 PL=0
MOVL C01781 V=800.0 PL=0
MOVL C01782 V=800.0 PL=0
MOVL C01783 V=800.0 PL=0
MOVL C01784 V=800.0 PL=0
MOVL C01785 V=800.0 PL=0
MOVL C01786 V=800.0 PL=0
MOVL C01787 V=800.0 PL=0
MOVL C01788 V=800.0 PL=0
MOVL C01789 V=800.0 PL=0
MOVL C01790 V=800.0 PL=0
MOVL C01791 V=800.0 PL=0
MOVL C01792 V=800.0 PL=0
MOVL C01793 V=800.0 PL=0
MOVL C01794 V=800.0 PL=0
MOVL C01795 V=800.0 PL=0
MOVL C01796 V=800.0 PL=0
MOVL C01797 V=800.0 PL=0
MOVL C01798 V=800.0 PL=0
MOVL C01799 V=800.0 PL=0
MOVL C01800 V=800.0 PL=0
MOVL C01801 V=800.0 PL=0
MOVL C01802 V=800.0 PL=0
MOVL C01803 V=800.0 PL=0
MOVL C01804 V=800.0 PL=0
MOVL C01805 V=800.0 PL=0
MOVL C01806 V=800.0 PL=0
MOVL C01807 V=800.0 PL=0
MOVL C01808 V=800.0 PL=0
MOVL C01809 V=800.0 PL=0
MOVL C01810 V=800.0 PL=0
MOVL C01811 V=800.0 PL=0
MOVL C01812 V=800.0 PL=0
MOVL C01813 V=800.0 PL=0
MOVL C01814 V=800.0 PL=0
MOVL C01815 V=800.0 PL=0
MOVL C01816 V=800.0 PL=0
MOVL C01817 V=800.0 PL=0
MOVL C01818 V=800.0 PL=0
MOVL C01819 V=800.0 PL=0
MOVL C01820 V=800.0 PL=0
MOVL C01821 V=800.0 PL=0
MOVL C01822 V=800.0 PL=0
MOVL C01823 V=800.0 PL=0
MOVL C01824 V=800.0 PL=0
MOVL C01825 V=800.0 PL=0
MOVL C01826 V=800.0 PL=0
MOVL C01827 V=800.0 PL=0
MOVL C01828 V=800.0 PL=0
MOVL C01829 V=800.0 PL=0
MOVL C01830 V=800.0 PL=0
MOVL C01831 V=800.0 PL=0
MOVL C01832 V=800.0 PL=0
MOVL C01833 V=800.0 PL=0
MOVL C01834 V=800.0 PL=0
MOVL C01835 V=800.0 PL=0
MOVL C01836 V=800.0 PL=0
MOVL C01837 V=800.0 PL=0
MOVL C01838 V=800.0 PL=0
MOVL C01839 V=800.0 PL=0
MOVL C01840 V=800.0 PL=0
MOVL C01841 V=800.0 PL=0
MOVL C01842 V=800.0 PL=0
MOVL C01843 V=800.0 PL=0
MOVL C01844 V=800.0 PL=0
MOVL C01845 V=800.0 PL=0
MOVL C01846 V=800.0 PL=0
MOVL C01847 V=800.0 PL=0
MOVL C01848 V=800.0 PL=0
MOVL C01849 V=800.0 PL=0
MOVL C01850 V=800.0 PL=0
MOVL C01851 V=800.0 PL=0
MOVL C01852 V=800.0 PL=0
MOVL C01853 V=800.0 PL=0
MOVL C01854 V=800.0 PL=0
MOVL C01855 V=800.0 PL=0
MOVL C01856 V=800.0 PL=0
MOVL C01857 V=800.0 PL=0
MOVL C01858 V=800.0 PL=0
MOVL C01859 V=800.0 PL=0
MOVL C01860 V=800.0 PL=0
MOVL C01861 V=800.0 PL=0
MOVL C01862 V=800.0 PL=0
MOVL C01863 V=800.0 PL=0
MOVL C01864 V=800.0 PL=0
MOVL C01865 V=800.0 PL=0
MOVL C01866 V=800.0 PL=0
MOVL C01867 V=800.0 PL=0
MOVL C01868 V=800.0 PL=0
MOVL C01869 V=800.0 PL=0
MOVL C01870 V=800.0 PL=0
MOVL C01871 V=800.0 PL=0
MOVL C01872 V=800.0 PL=0
MOVL C01873 V=800.0 PL=0
MOVL C01874 V=800.0 PL=0
MOVL C01875 V=800.0 PL=0
MOVL C01876 V=800.0 PL=0
MOVL C01877 V=800.0 PL=0
MOVL C01878 V=800.0 PL=0
MOVL C01879 V=800.0 PL=0
MOVL C01880 V=800.0 PL=0
MOVL C01881 V=800.0 PL=0
MOVL C01882 V=800.0 PL=0
MOVL C01883 V=800.0 PL=0
MOVL C01884 V=800.0 PL=0
MOVL C01885 V=800.0 PL=0
MOVL C01886 V=800.0 PL=0
MOVL C01887 V=800.0 PL=0
MOVL C01888 V=800.0 PL=0
MOVL C01889 V=800.0 PL=0
MOVL C01890 V=800.0 PL=0
MOVL C01891 V=800.0 PL=0
MOVL C01892 V=800.0 PL=0
MOVL C01893 V=800.0 PL=0
MOVL C01894 V=800.0 PL=0
MOVL C01895 V=800.0 PL=0
MOVL C01896 V=800.0 PL=0
MOVL C01897 V=800.0 PL=0
MOVL C01898 V=800.0 PL=0
MOVL C01899 V=800.0 PL=0
MOVL C01900 V=800.0 PL=0
MOVL C01901 V=800.0 PL=0
MOVL C01902 V=800.0 PL=0
MOVL C01903 V=800.0 PL=0
MOVL C01904 V=800.0 PL=0
MOVL C01905 V=800.0 PL=0
MOVL C01906 V=800.0 PL=0
MOVL C01907 V=800.0 PL=0
MOVL C01908 V=800.0 PL=0
MOVL C01909 V=800.0 PL=0
MOVL C01910 V=800.0 PL=0
MOVL C01911 V=800.0 PL=0
MOVL C01912 V=800.0 PL=0
MOVL C01913 V=800.0 PL=0
MOVL C01914 V=800.0 PL=0
MOVL C01915 V=800.0 PL=0
MOVL C01916 V=800.0 PL=0
MOVL C01917 V=800.0 PL=0
MOVL C01918 V=800.0 PL=0
MOVL C01919 V=800.0 PL=0
MOVL C01920 V=800.0 PL=0
MOVL C01921 V=800.0 PL=0
MOVL C01922 V=800.0 PL=0
MOVL C01923 V=800.0 PL=0
MOVL C01924 V=800.0 PL=0
MOVL C01925 V=800.0 PL=0
MOVL C01926 V=800.0 PL=0
MOVL C01927 V=800.0 PL=0
MOVL C01928 V=800.0 PL=0
MOVL C01929 V=800.0 PL=0
MOVL C01930 V=800.0 PL=0
MOVL C01931 V=800.0 PL=0
MOVL C01932 V=800.0 PL=0
MOVL C01933 V=800.0 PL=0
MOVL C01934 V=800.0 PL=0
MOVL C01935 V=800.0 PL=0
MOVL C01936 V=800.0 PL=0
MOVL C01937 V=800.0 PL=0
MOVL C01938 V=800.0 PL=0
MOVL C01939 V=800.0 PL=0
MOVL C01940 V=800.0 PL=0
MOVL C01941 V=800.0 PL=0
MOVL C01942 V=800.0 PL=0
MOVL C01943 V=800.0 PL=0
MOVL C01944 V=800.0 PL=0
MOVL C01945 V=800.0 PL=0
MOVL C01946 V=800.0 PL=0
MOVL C01947 V=800.0 PL=0
MOVL C01948 V=800.0 PL=0
MOVL C01949 V=800.0 PL=0
MOVL C01950 V=800.0 PL=0
MOVL C01951 V=800.0 PL=0
MOVL C01952 V=800.0 PL=0
MOVL C01953 V=800.0 PL=0
MOVL C01954 V=800.0 PL=0
MOVL C01955 V=800.0 PL=0
MOVL C01956 V=800.0 PL=0
MOVL C01957 V=800.0 PL=0
MOVL C01958 V=800.0 PL=0
MOVL C01959 V=800.0 PL=0
MOVL C01960 V=800.0 PL=0
MOVL C01961 V=800.0 PL=0
MOVL C01962 V=800.0 PL=0
MOVL C01963 V=800.0 PL=0
MOVL C01964 V=800.0 PL=0
MOVL C01965 V=800.0 PL=0
MOVL C01966 V=800.0 PL=0
MOVL C01967 V=800.0 PL=0
MOVL C01968 V=800.0 PL=0
MOVL C01969 V=800.0 PL=0
MOVL C01970 V=800.0 PL=0
MOVL C01971 V=800.0 PL=0
MOVL C01972 V=800.0 PL=0
MOVL C01973 V=800.0 PL=0
MOVL C01974 V=800.0 PL=0
MOVL C01975 V=800.0 PL=0
MOVL C01976 V=800.0 PL=0
MOVL C01977 V=800.0 PL=0
MOVL C01978 V=800.0 PL=0
MOVL C01979 V=800.0 PL=0
MOVL C01980 V=800.0 PL=0
MOVL C01981 V=800.0 PL=0
MOVL C01982 V=800.0 PL=0
MOVL C01983 V=800.0 PL=0
MOVL C01984 V=800.0 PL=0
MOVL C01985 V=800.0 PL=0
MOVL C01986 V=800.0 PL=0
MOVL C01987 V=800.0 PL=0
MOVL C01988 V=800.0 PL=0
MOVL C01989 V=800.0 PL=0
MOVL C01990 V=800.0 PL=0
MOVL C01991 V=800.0 PL=0
MOVL C01992 V=800.0 PL=0
MOVL C01993 V=800.0 PL=0
MOVL C01994 V=800.0 PL=0
MOVL C01995 V=800.0 PL=0
MOVL C01996 V=800.0 PL=0
MOVL C01997 V=800.0 PL=0
MOVL C01998 V=800.0 PL=0
MOVL C01999 V=800.0 PL=0
MOVL C02000 V=800.0 PL=0
MOVL C02001 V=800.0 PL=0
MOVL C02002 V=800.0 PL=0
MOVL C02003 V=800.0 PL=0
MOVL C02004 V=800.0 PL=0
MOVL C02005 V=800.0 PL=0
MOVL C02006 V=800.0 PL=0
MOVL C02007 V=800.0 PL=0
MOVL C02008 V=800.0 PL=0
MOVL C02009 V=800.0 PL=0
MOVL C02010 V=800.0 PL=0
MOVL C02011 V=800.0 PL=0
MOVL C02012 V=800.0 PL=0
MOVL C02013 V=800.0 PL=0
MOVL C02014 V=800.0 PL=0
MOVL C02015 V=800.0 PL=0
MOVL C02016 V=800.0 PL=0
MOVL C02017 V=800.0 PL=0
MOVL C02018 V=800.0 PL=0
MOVL C02019 V=800.0 PL=0
MOVL C02020 V=800.0 PL=0
MOVL C02021 V=800.0 PL=0
MOVL C02022 V=800.0 PL=0
MOVL C02023 V=800.0 PL=0
MOVL C02024 V=800.0 PL=0
MOVL C02025 V=800.0 PL=0
MOVL C02026 V=800.0 PL=0
MOVL C02027 V=800.0 PL=0
MOVL C02028 V=800.0 PL=0
MOVL C02029 V=800.0 PL=0
MOVL C02030 V=800.0 PL=0
MOVL C02031 V=800.0 PL=0
MOVL C02032 V=800.0 PL=0
MOVL C02033 V=800.0 PL=0
MOVL C02034 V=800.0 PL=0
MOVL C02035 V=800.0 PL=0
MOVL C02036 V=800.0 PL=0
MOVL C02037 V=800.0 PL=0
MOVL C02038 V=800.0 PL=0
MOVL C02039 V=800.0 PL=0
MOVL C02040 V=800.0 PL=0
MOVL C02041 V=800.0 PL=0
MOVL C02042 V=800.0 PL=0
MOVL C02043 V=800.0 PL=0
MOVL C02044 V=800.0 PL=0
MOVL C02045 V=800.0 PL=0
MOVL C02046 V=800.0 PL=0
MOVL C02047 V=800.0 PL=0
MOVL C02048 V=800.0 PL=0
MOVL C02049 V=800.0 PL=0
MOVL C02050 V=800.0 PL=0
MOVL C02051 V=800.0 PL=0
MOVL C02052 V=800.0 PL=0
MOVL C02053 V=800.0 PL=0
MOVL C02054 V=800.0 PL=0
MOVL C02055 V=800.0 PL=0
MOVL C02056 V=800.0 PL=0
MOVL C02057 V=800.0 PL=0
MOVL C02058 V=800.0 PL=0
MOVL C02059 V=800.0 PL=0
MOVL C02060 V=800.0 PL=0
MOVL C02061 V=800.0 PL=0
MOVL C02062 V=800.0 PL=0
MOVL C02063 V=800.0 PL=0
MOVL C02064 V=800.0 PL=0
MOVL C02065 V=800.0 PL=0
MOVL C02066 V=800.0 PL=0
MOVL C02067 V=800.0 PL=0
MOVL C02068 V=800.0 PL=0
MOVL C02069 V=800.0 PL=0
MOVL C02070 V=800.0 PL=0
MOVL C02071 V=800.0 PL=0
MOVL C02072 V=800.0 PL=0
MOVL C02073 V=800.0 PL=0
MOVL C02074 V=800.0 PL=0
MOVL C02075 V=800.0 PL=0
MOVL C02076 V=800.0 PL=0
MOVL C02077 V=800.0 PL=0
MOVL C02078 V=800.0 PL=0
MOVL C02079 V=800.0 PL=0
MOVL C02080 V=800.0 PL=0
MOVL C02081 V=800.0 PL=0
MOVL C02082 V=800.0 PL=0
MOVL C02083 V=800.0 PL=0
MOVL C02084 V=800.0 PL=0
MOVL C02085 V=800.0 PL=0
MOVL C02086 V=800.0 PL=0
MOVL C02087 V=800.0 PL=0
MOVL C02088 V=800.0 PL=0
MOVL C02089 V=800.0 PL=0
MOVL C02090 V=800.0 PL=0
MOVL C02091 V=800.0 PL=0
MOVL C02092 V=800.0 PL=0
MOVL C02093 V=800.0 PL=0
MOVL C02094 V=800.0 PL=0
MOVL C02095 V=800.0 PL=0
MOVL C02096 V=800.0 PL=0
MOVL C02097 V=800.0 PL=0
MOVL C02098 V=800.0 PL=0
MOVL C02099 V=800.0 PL=0
MOVL C02100 V=800.0 PL=0
MOVL C02101 V=800.0 PL=0
MOVL C02102 V=800.0 PL=0
MOVL C02103 V=800.0 PL=0
MOVL C02104 V=800.0 PL=0
MOVL C02105 V=800.0 PL=0
MOVL C02106 V=800.0 PL=0
MOVL C02107 V=800.0 PL=0
MOVL C02108 V=800.0 PL=0
MOVL C02109 V=800.0 PL=0
MOVL C02110 V=800.0 PL=0
MOVL C02111 V=800.0 PL=0
MOVL C02112 V=800.0 PL=0
MOVL C02113 V=800.0 PL=0
MOVL C02114 V=800.0 PL=0
MOVL C02115 V=800.0 PL=0
MOVL C02116 V=800.0 PL=0
MOVL C02117 V=800.0 PL=0
MOVL C02118 V=800.0 PL=0
MOVL C02119 V=800.0 PL=0
MOVL C02120 V=800.0 PL=0
MOVL C02121 V=800.0 PL=0
MOVL C02122 V=800.0 PL=0
MOVL C02123 V=800.0 PL=0
MOVL C02124 V=800.0 PL=0
MOVL C02125 V=800.0 PL=0
MOVL C02126 V=800.0 PL=0
MOVL C02127 V=800.0 PL=0
MOVL C02128 V=800.0 PL=0
MOVL C02129 V=800.0 PL=0
MOVL C02130 V=800.0 PL=0
MOVL C02131 V=800.0 PL=0
